*)
          
END_FUNCTION

FUNCTION RES_NTC : REAL
  VAR_INPUT
    T : REAL;
    RN : REAL;
    B : REAL;
  END_VAR

            RES_NTC := RN * EXP(B * (1.0 / (T+273.15) - 0.00335401643468053));



(* revision history

hm 30. dec. 2008	rev 1.0
	original version

hm	11. mar. 2009	rev 1.1
	changed real constants to use dot syntax

*)
          
END_FUNCTION

FUNCTION RES_PT : REAL
  VAR_INPUT
    T : REAL;
    R0 : REAL;
  END_VAR
  VAR CONSTANT
    A : REAL := 0.00390802;
    B : REAL := -5.802E-07;
    C : REAL := -4.2735E-12;
  END_VAR
  VAR
    T2 : REAL;
  END_VAR

            T2 := T * T;

IF T >= 0.0 THEN
	RES_PT := R0 * ( 1.0 + A * T + B * T2);
ELSE
	RES_PT := R0 * ( 1.0 + A * T + B * T2 + C * (T - 100.0) * T2 * T);
END_IF;



(* revision history
hm	4. aug. 2006	rev 1.1
	original version

hm	2. dec 2007	rev 1.2
	changed code for better performance

hm	11. mar. 2009	rev 1.3
	changed real constants to use dot syntax

*)


(*
 Auszug aus DIN 43760 für Pt100

°C		R		°C		R		°C	R			°C		R			°C		R			°C		R

-200 	18,49 	-100 	60,25 	0 	100,00 	100 	138,50 	200 	175,84 	300 	212,02
-195 	20,65 	-95 	62,28 	5 	101,95 	105 	140,39 	205 	177,68 	305 	213,80
-190 	22,80 	-90 	64,30 	10 	103,90 	110 	142,29 	210 	179,51 	310 	215,57
-185 	24,94 	-85 	66,31 	15 	105,85 	115 	144,17 	215 	181,34 	315 	217,35
-180 	27,08 	-80 	68,33 	20 	107,79 	120 	146,06 	220 	183,17 	320 	219,12
-175 	29,20 	-75 	70,33 	25 	109,73 	125 	147,94 	225 	184,99 	325 	220,88
-170 	31,32 	-70 	72,33 	30 	111,67 	130 	149,82 	230 	186,82 	330 	222,65
-165 	33,43 	-65 	74,33 	35 	113,61 	135 	151,70 	235 	188,63 	335 	224,41
-160 	35,33 	-60 	76,33 	40 	115,54 	140 	153,58 	240 	190,45 	340 	226,17
-155 	37,63 	-55 	78,32 	45 	117,47 	145 	155,45 	245 	192,26 	345 	227,92
-150 	39,71 	-50 	80,31 	50 	119,40 	150 	157,31 	250 	194,07 	350 	229,67
-145 	41,79 	-45 	82,29 	55 	121,32 	155 	159,18 	255 	195,88 	355 	231,42
-140 	43,87 	-40 	84,27 	60 	123,24 	160 	161,04 	260 	197,69 	360 	233,17
-135 	45,94 	-35 	86,25 	65 	125,16 	165 	162,90 	265 	199,49 	365 	234,91
-130 	48,00 	-30 	88,22 	70 	127,07 	170 	164,76 	270 	201,29 	370 	236,65
-125 	50,06 	-25 	90,19 	75 	128,98 	175 	166,61 	275 	203,08 	375 	238,39
-120 	52,11 	-20 	92,16 	80 	130,89 	180 	168,46 	280 	204,88 	380 	240,13
-115 	54,15 	-15 	94,12 	85 	132,80 	185 	170,31 	285 	206,67 	385 	241,86
-110 	56,19 	-10 	96,09 	90 	134,70 	190 	172,16 	290 	208,45 	390 	243,59
-105 	58,22 	-5 		98,04 	95 	136,60 	195 	174,00 	295 	210,24 	395 	245,31

*)
(*
revision history


*)
          
END_FUNCTION

FUNCTION RES_SI : REAL
  VAR_INPUT
    T : REAL;
    RS : REAL;
    TS : REAL;
  END_VAR
  VAR CONSTANT
    A : REAL := 0.00764;
    B : REAL := 1.66E-05;
  END_VAR
  VAR
    TX : REAL;
  END_VAR

            TX := T - TS;
RES_SI := RS * ( 1.0 + A * TX + B * TX * TX);

(* revision history
hm	4. aug 2006	rev 1.0
	original version

hm	2. dec 2007	rev 1.1
	changed code for better performance

hm	11. mar. 2009	rev 1.2
	changed real constants to use dot syntax

*)
          
END_FUNCTION

FUNCTION SENSOR_INT : REAL
  VAR_INPUT
    Voltage : REAL;
    Current : REAL;
    RP : REAL;
    RS : REAL;
  END_VAR
  VAR
    RG : REAL;
  END_VAR

            IF current <> 0.0 THEN
	RG := voltage / current;
	SENSOR_INT := RP * ( RG - RS) / ( RP + RS - RG);
END_IF;

(* revisaion history

hm 20.1.2007		rev 1.1
	deleted input R0 which was not needed.

hm	2. dec 2007	rev 1.2
	corrected an error in formula and improoved speed

hm	11. mar. 2009	rev 1.3
	changed real constants to use dot syntax

*)
          
END_FUNCTION

FUNCTION TEMP_NI : REAL
  VAR_INPUT
    Res : REAL;
    R0 : REAL;
  END_VAR

            TEMP_NI := (SQRT(0.30085225 - 2.66E-3 * (R0 - Res)) - 0.5485) * 751.8796992;


(* revision history

hm 24.1.2007		rev 1.1
	deleted unused variable A, B, C

hm 10.9.2007		rev 1.2
	changed accuracy to 0.02 degrees to improove performace

hm 17. 12 2007	rev 1.3
	improovements for better performance and higher accuracy

hm	6. jan 2008	rev 1.4
	further performance improvement

hm	10. mar. 2009	rev 1.5
	removed nested comments

*)


          
END_FUNCTION

FUNCTION TEMP_NTC : REAL
  VAR_INPUT
    RES : REAL;
    RN : REAL;
    B : REAL;
  END_VAR

            IF res > 0.0 THEN
	TEMP_NTC := B * 298.15 / (B + LN(RES / RN) * 298.15) -273.15;
END_IF;


(* revision history

hm 30. dec. 2008	rev 1.0
	original version

hm	11. mar. 2009	rev 1.1
	changed real constants to use dot syntax

*)
          
END_FUNCTION

FUNCTION TEMP_PT : REAL
  VAR_INPUT
    Res : REAL;
    R0 : REAL;
  END_VAR
  VAR CONSTANT
    A : REAL := 0.0039083;
    B : REAL := -5.775E-07;
    accuracy : REAL := 0.01;
  END_VAR
  VAR
    step : REAL := 50;
    X : REAL;
    Y : REAL;
    t1 : REAL;
    pt : POINTER TO DWORD;
  END_VAR

            X := A * R0;
Y := B * R0;
IF Res >= R0 THEN
	t1 := X * X - 4.0 * Y * (R0 - Res);
	IF t1 < 0.0 THEN
		TEMP_PT := 10000.0;
	ELSE
		TEMP_PT := (-X + SQRT(t1)) / (2.0 * Y);
	END_IF;
ELSE
	pt := ADR(step);
	(* since the formula cannot be solved this is a successive approximation *)
	TEMP_PT := -100.0;
	WHILE step > accuracy DO
		(* test if result greater or less *)
		IF RES_PT(TEMP_PT, R0) < res THEN TEMP_PT := TEMP_PT + step; ELSE TEMP_PT := TEMP_PT - step; END_IF;
		pt^ := pt^ - 8388608;  (* this is a super fast divide by 2 method for non floating point CPUs *)
		(* the alternative code: step := step * 0.5; *)
	END_WHILE;
END_IF;

(* revision history

rev 1.1 hm 24.1.2007	
	deleted unused variable C

rev 1.2 hm 10.9.2007
	reduced accuracy to 0.02 to shorten execution time

rev 1.3	hm	2. dec 2007
	changed code for better performance

rev	1.4	hm	23. dec 2007
	avoid a negative square root if input values are wrong

rev 1.5 hm	5. jan 2008
	replaced / 2 with * 0.5 for better performance

hm	31. oct. 2008	rev 1.6
	improved performance

hm	11. mar. 2009	rev 1.7
	changed real constants to use dot syntax

*)

          
END_FUNCTION

FUNCTION TEMP_SI : REAL
  VAR_INPUT
    Res : REAL;
    RS : REAL;
    TS : REAL;
  END_VAR

            TEMP_SI := (-7.64E-3 + SQRT(Res / RS * 6.64E-5 - 0.803E-5)) * 30120.48193 + TS;



(* revision history

hm 24.1.2007		rev 1.1
	the function would only work for TS = 25, now it works for other values of ts.

hm 10.9.2007		rev 1.2
	changed the function to use successive approcimation to avoid an error generated by a sqrt from a negative result.
	changed accuracy to 0.02 degrees to shorten execution time

hm 17. 12 2007	rev 1.3
	improovements for better performance

hm	6. jan 2008	rev 1.4
	further performance improvement

hm	10. mar. 2009	rev 1.5
	removed nested comments

*)
          
END_FUNCTION

FUNCTION_BLOCK _RMP_B
  VAR_INPUT
    DIR : BOOL;  (* true = up *)
    E : BOOL := TRUE;
    TR : TIME;
  END_VAR
  VAR_IN_OUT
    RMP : BYTE;
  END_VAR
  VAR
    tx : TIME;
    tl : TIME;
    tn : TIME;
    init : BOOL;
    last_dir : BOOL;
    start : BYTE;
  END_VAR

            (* read system timer *)
tx := DWORD_TO_TIME(T_PLC_MS());

IF E AND init AND (dir = last_dir) AND (RMP <> SEL(DIR, 0, 255)) AND TR = tn THEN
	RMP := FRMP_B(start, DIR, tx - tl, TR);
ELSE
	init := TRUE;
	tl := tx;
	tn := tr;
	start := RMP;
END_IF;
last_dir := dir;



(* revison history
hm	22. oct. 2008	rev 1.0
	original version

hm	20. nov. 2008	rev 1.1
	set default for E to be TRUE
	added init

hm	19. nov. 2011	rev 1.2
	new code
*)
          
END_FUNCTION_BLOCK

FUNCTION_BLOCK _RMP_NEXT
  VAR_INPUT
    E : BOOL := TRUE;
    IN : BYTE;
    TR : TIME;
    TF : TIME;
    TL : TIME;
  END_VAR
  VAR_OUTPUT
    DIR : BOOL;  (* upwards = TRUE *)
    UP : BOOL;
    DN : BOOL;
  END_VAR
  VAR_IN_OUT
    OUT : BYTE;
  END_VAR
  VAR
    rmx : _RMP_B;
    dirx : TREND_DW;
    t_lock : TP;
    xen : BOOL;
    xdir : BOOL;
  END_VAR

            dirx(X := in);

t_lock(in := FALSE, pt := TL);

IF dirx.TU AND (OUT < IN) THEN
	IF NOT xdir AND xen THEN t_lock(in := TRUE); END_IF;
	xen := TRUE;
	xdir := TRUE;
ELSIF dirx.TD AND (OUT > IN) THEN
	IF xdir AND xen THEN t_lock(in := TRUE); END_IF;
	xen := TRUE;
	xdir := FALSE;
ELSIF xen THEN
	IF (xdir AND (out >= in)) OR (NOT xdir AND (out <= in)) THEN
		xen := FALSE;
		IF tl > t#0s THEN t_lock(IN := TRUE); END_IF;
	END_IF;
END_IF;

IF NOT t_lock.Q AND xen THEN
		UP := XDIR;
		DIR := XDIR;
		DN := NOT XDIR;
ELSE
	UP := FALSE;
	DN := FALSE;
END_IF;

rmx(rmp := OUT, E := E AND (UP OR DN) , dir := DIR, tr := SEL(dir, TF, TR));


(* revison history
hm	23. nov. 2008	rev 1.0
	original version

hm	24. jan. 2009	rev 1.1
	deleted unused vars tmp1, tmp2

hm	20. feb. 2009	rev 1.2
	improved algorithm
	added TL

hm	9. mar. 2009	rev 1.3
	input E was ignored
	removed double assignments

hm	18. jul. 2009	rev 1.4
	improved performance

*)
          
END_FUNCTION_BLOCK

FUNCTION_BLOCK _RMP_W
  VAR_INPUT
    DIR : BOOL;
    E : BOOL := TRUE;
    TR : TIME;
  END_VAR
  VAR_IN_OUT
    RMP : WORD;
  END_VAR
  VAR
    tx : DWORD;
    tl : DWORD;
    step : DINT;
    init : BOOL;
    last_dir : BOOL;
  END_VAR

            tx := T_PLC_MS();
IF E AND init THEN
	(* we need to set tl = tx when direction changes *)
	IF dir XOR last_dir THEN
	 tl := tx;
	 last_dir := dir;
	END_IF;
	(* check_elapsed time and calculate only if necessary *)
	IF tr > t#0s THEN
		step := DWORD_TO_DINT(SHL(tx-tl, 16) / TIME_TO_DWORD(TR));
	ELSE
		step := 65535;
	END_IF;
	IF step > 0 THEN
		(* perform the step on the ramp *)
		tl := tx;
		(* calculate the step response *)
		IF NOT dir THEN step := - step; END_IF;
		rmp := DINT_TO_WORD(LIMIT(0, WORD_TO_DINT(rmp) + step, 65535));
	END_IF;
ELSE
	tl := tx;
	init := TRUE;
END_IF;


(* revison history
hm	22. oct. 2008	rev 1.0
	original version

hm	20. nov. 2008	rev 1.1
	set default for E to be TRUE
	added init

*)
          
END_FUNCTION_BLOCK

FUNCTION_BLOCK GEN_PULSE
  VAR_INPUT
    ENQ : BOOL := TRUE;
    PTH : TIME;
    PTL : TIME;
  END_VAR
  VAR_OUTPUT
    Q : BOOL;
  END_VAR
  VAR
    tx : TIME;
    tn : TIME;
    init : BOOL;
  END_VAR

            
IF enq THEN
	tx := DWORD_TO_TIME(T_PLC_MS());
	IF NOT init THEN init := TRUE; tn := tx; END_IF;
	IF tx - tn >= SEL(Q, PTL, PTH) THEN
		Q := NOT Q;
		tn := tn + SEL(Q, PTL, PTH);
	END_IF;
ELSE
	Q := FALSE;
	init := FALSE;
END_IF;


(* revision history
hm	29. jun. 2008	rev 1.0
	original version

hm	23. nov. 2008	rev 1.1
	set default for enq to be true

hm	18. jul. 2009	rev 1.2
	improved performance

hm	13. nov. 2009	rev 1.3
	corrected error

hm	16. feb. 2011	rev 1.4
	corrected an error when timer overflows

*)
          
END_FUNCTION_BLOCK

FUNCTION_BLOCK GEN_PW2
  VAR_INPUT
    ENQ : BOOL;
    TH1 : TIME;
    TL1 : TIME;
    TH2 : TIME;
    TL2 : TIME;
    TS : BOOL;
  END_VAR
  VAR_OUTPUT
    Q : BOOL;
    TH : TIME;
    TL : TIME;
  END_VAR
  VAR
    t_high : TIME;
    t_low : TIME;
    tx : TIME;
    start : TIME;
    init : BOOL;
    et : TIME;
  END_VAR

            (* read system timer *)
tx := DWORD_TO_TIME(T_PLC_MS());

(* startup initialization *)
IF NOT init THEN
	start := tx;
	init := TRUE;
	TH := T#0s;
	TL := T#0s;
END_IF;

(* timing selection *)
IF TS THEN
	t_high := TH2;
	t_low := TL2;
ELSE
	t_high := TH1;
	t_low := TL1;
END_IF;

(* normal operation *)
IF ENQ THEN
	et := tx - start;
	IF NOT Q THEN
		IF et >= t_low THEN
			Q := TRUE;
			start := tx;
			TL := T#0s;
		ELSE
			TL := et;
		END_IF;
	ELSE
		IF et >= t_high THEN
			Q := FALSE;
			start := tx;
			TH := T#0s;
		ELSE
			TH := et;
		END_IF;
	END_IF;
ELSE
	Q := FALSE;
	TH := T#0s;
	TL := T#0s;
	start := tx;
END_IF;



(* revision history
hm	26. sep. 2008	rev 1.0
	original version

hm	14. mar. 2009	rev 1.1
	removed double assignments

*)
          
END_FUNCTION_BLOCK

FUNCTION_BLOCK GEN_RDM
  VAR_INPUT
    PT : TIME;
    AM : REAL := 1;
    OS : REAL;
  END_VAR
  VAR_OUTPUT
    Q : BOOL;
    Out : REAL;
  END_VAR
  VAR
    tx : TIME;
    last : TIME;
    init : BOOL;
  END_VAR

            (* read system time and prepare input data *)
tx := DWORD_TO_TIME(T_PLC_MS()) - last;

(* init section *)
IF NOT init THEN
	init := TRUE;
	last := tx;
	tx := t#0s;
END_IF;

(* add last if one cycle is finished *)
IF tx >= pt THEN
	last := last + pt;
	tx := tx - pt;

	(* generate output signal *)
	out := am * (RDM(0) - 0.5) + os;
	q := TRUE;
ELSE
	q := FALSE;
END_IF;

(* revision history

hm	7.2.2007		rev 1.0
	original version

hm	16.9.2007		rev 1.1
	changes time() to T_plc_ms() for compatibility reasons

*)

          
END_FUNCTION_BLOCK

FUNCTION_BLOCK GEN_RDT
  VAR_INPUT
    Enable : BOOL := TRUE;
    Min_Time_ms : TIME := TIME#1s0ms;  (* min Taktzeit *)
    Max_Time_ms : TIME := TIME#1s200ms;  (* Max Taktzeit *)
    TP_Q : TIME := TIME#100ms;  (* Zeit Ausgang auf TRUE *)
  END_VAR
  VAR_OUTPUT
    xQ : BOOL;
  END_VAR
  VAR
    tonRDMTimer : TON;  (* Zeitbaustein Taktgenerator *)
    tof_xQ : TOF;  (* Ausschaltverzögerung Taktgenerator *)
    tRDMTime : TIME;  (* Sollzeit *)
    rRDMTime : REAL;  (* Zufalswert Timer *)
  END_VAR

            tonRDMTimer ( IN:= Enable , PT:= tRDMTime );
tof_xQ ( IN:= tonRDMTimer.Q , PT:= TP_Q );
XQ := tof_xq.Q;
IF tonRDMTimer.Q THEN
		 xQ := TRUE ;
		 rRDMTime := RDM ( last:= rRDMTime ) ;
		 tRDMTime := REAL_TO_TIME ( rRDMTime * DINT_TO_REAL(TIME_TO_DINT( Max_Time_ms - Min_Time_ms ) + TIME_TO_DINT(Min_Time_ms ))) ;
		 tonRDMTimer ( IN:= FALSE );
END_IF;

(* revision history
J. Schohaus	19. nov 2007	rev 1.0
	origial version

hm	16. mar. 2008			rev 1.1
	added type conversion to avoid warnings under codesys 3.0
*)
          
END_FUNCTION_BLOCK

FUNCTION_BLOCK GEN_RMP
  VAR_INPUT
    PT : TIME := TIME#1s0ms;
    AM : REAL := 1;
    OS : REAL;
    DL : REAL;
  END_VAR
  VAR_OUTPUT
    Q : BOOL;
    OUT : REAL;
  END_VAR
  VAR
    tx : TIME;
    last : TIME;
    init : BOOL;
    temp : REAL;
    ltemp : REAL;
  END_VAR

            (* read system time and prepare input data *)
tx := DWORD_TO_TIME(T_PLC_MS()) - last;
DL := MODR(dl,1.0);
IF dl < 0.0 THEN dl := 1.0 - dl; END_IF;

(* init section *)
IF NOT init THEN
	init := TRUE;
	last := tx;
	tx := t#0s;
END_IF;

(* add last if one cycle is finished *)
IF tx >= pt THEN
	last := last + pt;
	tx := tx - pt;
END_IF;

(* generate sine wave *)
ltemp := temp;
IF pt > t#0s THEN temp := FRACT(TIME_TO_REAL(tx + MULTIME(pt, dl)) / TIME_TO_REAL(pt)); END_IF;
out := am * temp + os;

(* boolean output Q *)
Q := temp < ltemp;

(* revision history
hm	3. mar 2007		rev 1.0
	original version

hm	17 sep 2007		rev 1.1
	replaced time() with t_plc_ms for compatibilitx reasons

hm	27. nov 2007	rev 1.2
	avoid divide by 0 when pt = 0

ks	26. oct. 2008	rev 1.3
	code optimization

hm	10. mar. 2009	rev 1.4
	changed real constants to use dot syntax
*)
          
END_FUNCTION_BLOCK

FUNCTION_BLOCK GEN_SIN
  VAR_INPUT
    PT : TIME;
    AM : REAL := 1;
    OS : REAL;
    DL : REAL;
  END_VAR
  VAR_OUTPUT
    Q : BOOL;
    Out : REAL;
  END_VAR
  VAR
    tx : TIME;
    last : TIME;
    init : BOOL;
    temp : REAL;
  END_VAR

            (* read system time and prepare input data *)
tx := DWORD_TO_TIME(T_PLC_MS()) - last;
DL := MODR(dl,1.0);
IF dl < 0.0 THEN dl := 1.0 - dl; END_IF;

(* init section *)
IF NOT init THEN
	init := TRUE;
	last := tx;
	tx := t#0s;
END_IF;

(* add last if one cycle is finished *)
IF tx >= pt THEN
	last := last + pt;
	tx := tx - pt;
END_IF;

(* generate sine wave *)
IF pt > t#0s THEN temp := SIN(math.PI2 * DWORD_TO_REAL(TIME_TO_DWORD(tx + MULTIME(pt, dl))) / DWORD_TO_REAL(TIME_TO_DWORD(pt))); END_IF;
out := am * 0.5 *  temp + os;

(* boolean output Q *)
q := NOT SIGN_R(temp);

(* revision history
hm	22. jan 2007	rev 1.0
	original version

hm	17 sep 2007	rev 1.1
	replaced time() with t_plc_ms for compatibilitx reasons

hm	27. nov 2007	rev 1.2
	avoid divide by 0 when pt = 0

hm	6. jan 2008		rev 1.3
	improved performance

hm	16. mar. 2008	rev 1.4
	added type conversion to avoid warnings under codesys 3.0

hm	18. oct. 2008	rev 1.5
	using math constants

hm	11. mar. 2009	rev 1.6
	changed real constants to use dot syntax

*)
          
END_FUNCTION_BLOCK

FUNCTION_BLOCK GEN_SQR
  VAR_INPUT
    PT : TIME;
    AM : REAL := 1;
    OS : REAL;
    DC : REAL := 0.5;
    DL : REAL;
  END_VAR
  VAR_OUTPUT
    Q : BOOL;
    Out : REAL;
  END_VAR
  VAR
    tx : TIME;
    last : TIME;
    init : BOOL;
  END_VAR

            (* check dc = 1 or 0 *)
IF dc = 0.0 THEN
	out := -am * 0.5 + os;
	Q := FALSE;
	RETURN;
ELSIF dc = 1.0 THEN
	out := am * 0.5 + os;
	Q := TRUE;
	RETURN;
END_IF;

(* read system time and prepare input data *)
tx := DWORD_TO_TIME(T_PLC_MS()) - last;
DL := MODR(dl,1.0);
IF dl < 0.0 THEN dl := 1.0 - dl; END_IF;
dc := MODR(dc,1.0);
IF dc < 0.0 THEN dc := 1.0 - dc; END_IF;

(* init section *)
IF NOT init THEN
	init := TRUE;
	last := tx;
	tx := t#0s;
END_IF;

(* add last if one cycle is finished *)
IF tx >= pt THEN
	last := last + pt;
	tx := tx - pt;
END_IF;

(* check if falling or rising edge first *)
IF MULTIME(pt, dl + dc) >= pt THEN
	(* generate falling edge *)
	IF tx >= MULTIME(pt, dl + dc - 1) THEN
		out := -am * 0.5 + os;
		Q := FALSE;
	END_IF;
	(* generate rising edge *)
	IF tx >= MULTIME(pt, dl) THEN
		out := am * 0.5 + os;
		Q := TRUE;
	END_IF;
ELSE
	(* generate rising edge first *)
	IF tx >= MULTIME(pt, dl) THEN
		out := am * 0.5 + os;
		Q := TRUE;
	END_IF;
	(* generate falling edge *)
	IF tx >= MULTIME(pt, dl + dc) THEN
		out := -am * 0.5 +os;
		Q := FALSE;
	END_IF;
END_IF;

(* revision history

hm	12. feb 2007	rev 1.1
	added default value for dc = 0.5

hm	17 sep 2007	rev 1.2
	replaced time() with t_plc_ms for compatibilitx reasons

hm	6. jan 2008	rev 1.3
	improved performance

hm	11. mar. 2009	rev 1.4
	changed real constants to use dot syntax
	set default amplitude to 1.0

*)

          
END_FUNCTION_BLOCK

FUNCTION_BLOCK PWM_DC
  VAR_INPUT
    F : REAL;
    DC : REAL;
  END_VAR
  VAR_OUTPUT
    Q : BOOL;
  END_VAR
  VAR
    clk : CLK_PRG;
    pulse : TP_X;
    tmp : REAL;
  END_VAR

            IF F > 0.0 THEN
	tmp := 1000.0 / F;
	CLK(PT := REAL_TO_TIME(tmp));
	Pulse(in := clk.Q, pt := REAL_TO_TIME(tmp * DC));
	Q := pulse.Q;
END_IF;

(* revision history

hm	25. feb 2007	rev 1.1
	recoded in st for better performance and better portability

hm	27. nov 2007	rev 1.2
	avoid divide by 0 when F = 0

hm	19. oct. 2008	rev 1.3
	changed type TP_R to TP_X because of name change
	improved performance

hm	11. mar. 2009	rev 1.4
	changed real constants to use dot syntax

*)
          
END_FUNCTION_BLOCK

FUNCTION_BLOCK PWM_PW
  VAR_INPUT
    F : REAL;
    PW : TIME;
  END_VAR
  VAR_OUTPUT
    Q : BOOL;
  END_VAR
  VAR
    clk : CLK_PRG;
    pulse : TP_X;
  END_VAR

            IF F > 0.0 THEN
	CLK(PT := REAL_TO_TIME(1000.0 / F));
	Pulse(in := clk.Q, pt := pw);
	Q := pulse.Q;
END_IF;

(* revision history

hm	25. feb 2007	rev 1.1
	recoded in st for better performance and better portability

hm	27. nov 2007	rev 1.2
	avoid divide by 0 when F = 0

hm	9. dec 2007		rev 1.3
	corrected an error with F = 0

hm	19. oct. 2008	rev 1.4
	changed type tp_r to TP_x brecause of name change

hm	11. mar. 2009	rev 1.5
	changed real constants to use dot syntax

*)
          
END_FUNCTION_BLOCK

FUNCTION_BLOCK RMP_B
  VAR_INPUT
    SET : BOOL;
    PT : TIME;
    E : BOOL := TRUE;
    UP : BOOL := TRUE;
    RST : BOOL;
  END_VAR
  VAR_OUTPUT
    OUT : BYTE;
    BUSY : BOOL;
    HIGH : BOOL;
    LOW : BOOL;
  END_VAR
  VAR
    rmp : _RMP_B;
  END_VAR

            (* generate ramp *)
rmp(dir := UP, E := E, TR := PT, rmp := out);

(* set or reset operation *)
IF RST THEN
	out := 0;
ELSIF SET THEN
	out := 255;
END_IF;

(* checks for outputs stable and reset or set busy flag *)
low := out = 0;
high := out = 255;
busy := NOT (low OR high) AND E;


(* revision history

hm 5.10.2006	rev 1.1
	added busy output
hm 17.1.2007	rev 1.2
	renamed input ud to up for better usability
	deleted unused variable step

hm	17.9.2007		rev 1.3
	replaced time() with t_plc_ms() for compatibility reasons

hm	28. sep 2007	rev 1.4
	added outputs on and off
	busy is now disabled while en is false
	new coding for higher accuracy and performance

hm	5. oct 2007	rev 1.5
	added statements to allow for PT to be t#0s output jumps to max or min immediately

hm	25. dec 2007	rev 1.6
	improved code for better performance

hm	16. oct. 2008	rev 1.7
	improved code for better performance

hm	18. oct. 2008	rev 1.8
	added type conversion to avoid warnings
	changed input en to e for compatibility reasons

hm	23. oct. 2008	REV 	2.0
	new code using _RMP_B

*)
          
END_FUNCTION_BLOCK

FUNCTION_BLOCK RMP_SOFT
  VAR_INPUT
    IN : BOOL;
    VAL : BYTE;
    {attribute 'input_constant'}
    PT_ON : TIME;
    {attribute 'input_constant'}
    PT_OFF : TIME;
  END_VAR
  VAR_OUTPUT
    OUT : BYTE;
  END_VAR
  VAR
    rmp : _RMP_B;
    tmp : BYTE;
  END_VAR

            tmp := SEL(in, 0, val);
IF tmp > out THEN
	(* we need to ramp down *)
	rmp(dir := TRUE, E := TRUE, TR := PT_ON, rmp := out);
	(* make sure out does not surpass tmp *)
	out := MIN(out, tmp);
ELSIF tmp < out THEN
	(* we need to ramp up *)
	rmp(dir := FALSE, E := TRUE, TR := PT_OFF, rmp := out);
	(* make sure out does not surpass tmp *)
	out := MAX(out, tmp);
ELSE
	(* no ramp necessary *)
	rmp(E := FALSE, rmp := out);
END_IF;


(* revision history

hm 22.1.2007	rev 1.1
	deleted unused variables X1 and I, X2 and X3

hm	17.9.2007	rev 1.2
	replaced time() with t_plc_ms() for compatibility reasons

hm	26. oct. 2008	2.0
	new code using _rmp_b
*)

          
END_FUNCTION_BLOCK

FUNCTION_BLOCK RMP_W
  VAR_INPUT
    SET : BOOL;
    PT : TIME;
    E : BOOL := TRUE;
    UP : BOOL := TRUE;
    RST : BOOL;
  END_VAR
  VAR_OUTPUT
    out : WORD;
    busy : BOOL;
    high : BOOL;
    low : BOOL;
  END_VAR
  VAR
    rmp : _RMP_W;
  END_VAR

            (* generate ramp *)
rmp(dir := UP, E := E, TR := PT, rmp := out);

(* set or reset operation *)
IF RST THEN
	out := 0;
ELSIF SET THEN
	out := 65535;
END_IF;

(* checks for outputs stable and reset or set busy flag *)
low := out = 0;
high := out = 65535;
busy := NOT (low OR high) AND E;


(* revision history:

hm 4.10.2006		rev 1.1
	added the busy output which signals that the ramp is running.

hm 22.1.2007		rev 1.2
	deleted unused variable step

hm	17.9.2007		rev 1.3
	replaced time() with t_plc_ms() for compatibility reasons

hm	28. sep 2007	rev 1.4
	added outputs on and off
	busy is now disabled while en is false
	new coding for higher accuracy and performance

hm	5. oct 2007	rev 1.5
	added statements to allow for PT to be t#0s output jumps to max or min immediately

hm	2. dec 2007	rev 1.6
	corrected an error in calculation of step response

hm	25. dec 2007	rev 1.7
	corrected an error while step response was too slow for fast rise times

hm	16. oct. 2008	rev 1.8
	improved performance

hm	18. oct. 2008	rev 1.9
	renamed inout EN to E for compatibility reasons

hm	23. oct. 2008	rev 2.0
	new code using _RMP_W
*)

          
END_FUNCTION_BLOCK

FUNCTION AIN : REAL
  VAR_INPUT
    in : DWORD;
    {attribute 'input_constant'}
    Bits : BYTE;
    {attribute 'input_constant'}
    sign : BYTE := 255;
    {attribute 'input_constant'}
    low : REAL;
    {attribute 'input_constant'}
    high : REAL := 10;
  END_VAR
  VAR CONSTANT
    ff : DWORD := 16#FFFFFFFF;
  END_VAR
  VAR
    temp1 : DWORD;
    temp2 : DWORD;
    sx : BOOL;
  END_VAR

            (* extract the sign bit *)
IF sign < 32 THEN
	temp1 := SHR(in,sign);
	sx := temp1.0;
ELSE
	sx := FALSE;
END_IF;
temp1 := SHR(ff, 32-bits);
temp2 := in AND temp1;
AIN := (high - low) * DWORD_TO_REAL(temp2) / DWORD_TO_REAL(temp1) + low;
IF sx THEN AIN := -AIN; END_IF;

(* revision history
hm 18.8.2006	rev 1.1
	fixed an error with low value negative and high value 0.

hm 19.1.2007	rev 1.2
	fixed an error with sign bit.

hm	13.9.2007	rev 1.3
	changed code to avoid warning under codesys 2.8.1

hm	2. dec 2007	rev 1.4
	changed code for better performance

hm	16. mar 2008	rev 1.5
	added type conversions to avoid warnings under codesys 30
*)
          
END_FUNCTION

FUNCTION_BLOCK AIN1
  VAR_INPUT
    in : DWORD;
    {attribute 'input_constant'}
    sign_bit : INT := 255;
    {attribute 'input_constant'}
    error_bit : INT := 255;
    {attribute 'input_constant'}
    error_code_en : BOOL;
    {attribute 'input_constant'}
    error_code : DWORD;
    {attribute 'input_constant'}
    overflow_bit : INT := 255;
    {attribute 'input_constant'}
    overflow_code_en : BOOL;
    {attribute 'input_constant'}
    overflow_code : DWORD;
    {attribute 'input_constant'}
    Bit_0 : INT;
    {attribute 'input_constant'}
    Bit_N : INT := 31;
    {attribute 'input_constant'}
    out_min : REAL;
    {attribute 'input_constant'}
    out_max : REAL := 10;
    {attribute 'input_constant'}
    code_min : DWORD;
    {attribute 'input_constant'}
    code_max : DWORD := 16#FFFFFFFF;
    {attribute 'input_constant'}
    error_output : REAL;
    {attribute 'input_constant'}
    overflow_output : REAL := 10;
  END_VAR
  VAR_OUTPUT
    out : REAL;
    sign : BOOL;
    error : BOOL;
    overflow : BOOL;
  END_VAR
  VAR
    tB : DWORD;
  END_VAR

            (* extract error bit *)
error := ((SHR(in,error_bit) AND 16#0000_0001) = 1) OR (error_code_en AND error_code = in);
IF error THEN
	out := error_output;
	RETURN;
END_IF;

(* strip off the data input *)
tb := SHR(SHL(in, 31 - bit_N), 31 - bit_N + Bit_0);

(* extract overflow bit *)
overflow := ((SHR(in,overflow_bit) AND 16#0000_0001) = 1) OR (overflow_code_en AND overflow_code = in) OR (tb < code_min OR tb > code_max);
IF overflow THEN
	out := overflow_output;
	RETURN;
END_IF;

(* extract sign bit *)
sign := (SHR(in,sign_bit) AND 16#0000_0001) = 1;

(* convert in to out *)
out := (DWORD_TO_REAL(tb - code_min) * (out_max - out_min) / DWORD_TO_REAL(code_max - code_min) + out_min);
IF sign THEN out := out * -1.0; END_IF;



(* revision history
hm	23. feb 2008	rev 1.0
	original version

hm	16. mar 2008	rev 1.1
	added type conversions to avoid warnngs under codesys 30

hm	22. apr. 2008	rev 1.2
	corrected error in formula when code_min was set
	corrected error when sign bit was used
	optimized code for better performance

hm	10. mar. 2009	rev 1.3
	real constants updated to new systax using dot

*)
          
END_FUNCTION_BLOCK

FUNCTION AOUT : DWORD
  VAR_INPUT
    in : REAL;
    {attribute 'input_constant'}
    Bits : BYTE;
    {attribute 'input_constant'}
    sign : BYTE := 255;
    {attribute 'input_constant'}
    low : REAL;
    {attribute 'input_constant'}
    high : REAL := 10;
  END_VAR
  VAR CONSTANT
    ff : DWORD := 2#1;
  END_VAR
  VAR
    in2 : REAL;
    sx : BOOL;
  END_VAR

            (* if sign bit is defined *)
IF sign < 32 THEN
	sx := sign_R(in);
	in2 := ABS(in);
ELSE
	in2 := in;
END_IF;

(* begrenze in auf die zulässigen werte *)
in2 := LIMIT(low, in2, high);

(* Berechne den Ausgangswert *)
Aout := REAL_TO_DWORD((in2 - low) / (high - low) * DWORD_TO_REAL(SHL(ff,bits) -1));
IF sx THEN Aout := SHL(ff,sign) OR Aout; END_IF;

(*
revision history

hm 18.1.2007		rev 1.1
	renamed Modul to aout.
	changed Output to 32 Bit max.
	corrected error with sign bit.

hm	13.9.2007		rev 1.2
	changed code to avoid warning under codesys 2.8.1

hm	2. dec 2007		rev 1.3
	changed code for better performance

hm	23. feb 2008	rev 1.4
	changed code for better performance
*)
          
END_FUNCTION

FUNCTION AOUT1 : DWORD
  VAR_INPUT
    in : REAL;
    {attribute 'input_constant'}
    Bit_0 : INT;
    {attribute 'input_constant'}
    Bit_N : INT := 31;
    {attribute 'input_constant'}
    sign : INT := 255;
    {attribute 'input_constant'}
    low : REAL;
    {attribute 'input_constant'}
    high : REAL := 10;
  END_VAR
  VAR CONSTANT
    ff : DWORD := 2#1;
  END_VAR
  VAR
    sx : BOOL;
    in2 : REAL;
  END_VAR

            (* if sign bit is defined *)
IF sign < 32 THEN
	sx := SIGN_R(in);
	in2 := ABS(in);
ELSE
	in2 := in;
END_IF;

(* begrenze in auf die zulässigen werte *)
in2 := LIMIT(low, in2, high);

(* Berechne den Ausgangswert *)
AOUT1 := SHL(REAL_TO_DWORD((in2 - low) / (high - low) * DWORD_TO_REAL(SHL(ff,bit_n - Bit_0 + 1) -1)),Bit_0);
IF sx THEN AOUT1 := SHL(ff,sign) OR AOUT1; END_IF;


(* revision history
hm	23. feb 2008	rev 1.0
	original version

*)
          
END_FUNCTION

FUNCTION BYTE_TO_RANGE : REAL
  VAR_INPUT
    X : BYTE;
    low : REAL;
    high : REAL;
  END_VAR

            BYTE_TO_RANGE := (high - low) * X / 255.0 + low;


(* revision history
hm	9. jan 2008		rev 1.0
	original version

*)

          
END_FUNCTION

FUNCTION_BLOCK DELAY
  VAR_INPUT
    IN : REAL;
    N : INT;
    RST : BOOL;
  END_VAR
  VAR_OUTPUT
    OUT : REAL;
  END_VAR
  VAR
    buf : ARRAY[0..31] OF REAL;
    i : INT;
    init : BOOL;
    stop : INT;
  END_VAR

            stop := LIMIT(0,N,32) - 1;
IF rst OR NOT init THEN
	init := TRUE;
	FOR i := 0 TO stop DO buf[i] := in; END_FOR;
	out := in;
	i := 0;
ELSIF stop < 0 THEN
	out := in;
ELSE
	out := buf[i];
	buf[i] := in;
	i := INC1(i, N);
END_IF;



(* revision history
hm 1.10.2006		rev 1.1
	corrected error in buffer management

hm 19.1.2007		rev 1.2
	changed reset to load the value of in instead of 0

hm	27. oct. 2008	rev 1.3
	improved performance

hm	23. feb.2009	rev 1.4
	corrected an index problem

hm	23. mar. 2009	rev 1.5
	corrected non standard write to input N

*)
          
END_FUNCTION_BLOCK

FUNCTION_BLOCK DELAY_4
  VAR_INPUT
    in : REAL;
  END_VAR
  VAR_OUTPUT
    out1 : REAL;
    out2 : REAL;
    out3 : REAL;
    out4 : REAL;
  END_VAR
  VAR
    temp : REAL;
  END_VAR

            out4 := out3;
out3 := out2;
out2 := out1;
out1 := temp;
temp := in;

(* revision history

hm 19.1.2007	rev 1.1
	added variable temp to add 1 delay  for q1

*)
          
END_FUNCTION_BLOCK

FUNCTION_BLOCK FADE
  VAR_INPUT
    IN1 : REAL;
    IN2 : REAL;
    F : BOOL;
    TF : TIME;
    rst : BOOL;
  END_VAR
  VAR_OUTPUT
    Y : REAL;
  END_VAR
  VAR
    rmx : RMP_W;
  END_VAR

            rmx(rst := rst AND NOT F, set := rst AND F, pt := TF, up := F);
Y := (in2 - In1) / 65535.0 * WORD_TO_REAL(rmx.out) + in1;


(* code for rev 1.1
IF rst THEN
	rmx(set := F, rst := NOT F);
ELSIF F AND (NOT rmx.high) THEN
	rmx(PT := TF, UP := TRUE, e := TRUE, rst := FALSE, set := FALSE);
ELSIF (NOT F) AND (NOT rmx.low) THEN
	rmx(PT := TF, UP := FALSE, e := TRUE, rst := FALSE, set := FALSE);
ELSE
	rmx(e := FALSE, rst := FALSE, set := FALSE);
END_IF;
Y := (WORD_TO_REAL(rmx.out) * in1 + WORD_TO_REAL(FF - rmx.out) * IN2) / FF;
*)


(* revision history
hm	26. dec 2007	rev 1.0
	original version

hm	18. oct. 2008	rev 1.1
	improved performance
	changed calls for rmp_w because rmp_w has chaged

hm	17. dec. 2008	rev 1.2
	function of input f was inverted

hm	24. jan. 2009	rev 1.3
	delted unused var FF
*)
          
END_FUNCTION_BLOCK

FUNCTION_BLOCK FILTER_DW
  VAR_INPUT
    X : DWORD;
    T : TIME;
  END_VAR
  VAR_OUTPUT
    Y : DWORD;
  END_VAR
  VAR
    last : DWORD;
    tx : DWORD;
    init : BOOL;
    Yi : REAL;
  END_VAR

            (* read system time *)
tx := T_PLC_MS();

(* startup initialisation *)
IF NOT init OR T = t#0s THEN
	init := TRUE;
	Yi := DWORD_TO_REAL(X);
ELSE
	Yi := Yi + (DWORD_TO_REAL(X) - DWORD_TO_REAL(Y)) * DWORD_TO_REAL(tx - last) / TIME_TO_REAL(T);
END_IF;
last := tx;

Y := REAL_TO_DWORD(Yi);



(*
hm 10. oct. 2008	rev 1.0
	original version

hm	3. nov. 2008	REV 1.1
	corrected an overflow problem
*)
          
END_FUNCTION_BLOCK

FUNCTION_BLOCK FILTER_I
  VAR_INPUT
    X : INT;
    T : TIME;
  END_VAR
  VAR_OUTPUT
    Y : INT;
  END_VAR
  VAR
    Yi : DINT;
    last : DWORD;
    tx : DWORD;
    init : BOOL;
  END_VAR

            (* read system time *)
tx := T_PLC_MS();

(* startup initialisation *)
IF NOT init OR T = t#0s THEN
	init := TRUE;
	Yi := INT_TO_DINT(X) * 1000;
ELSE
	(* to increase accuracy of the filter we calculate internal Yi wich is Y * 1000 *)
	Yi := Yi + INT_TO_DINT(X - Y) * DWORD_TO_DINT(tx - last) * 1000 / TIME_TO_DINT(T);
END_IF;
last := tx;
Y := DINT_TO_INT(yi / 1000);



(*
hm 8. nov. 2008	rev 1.0
	original version

*)
          
END_FUNCTION_BLOCK

FUNCTION_BLOCK FILTER_MAV_DW
  VAR_INPUT
    X : DWORD;
    N : UINT;
    RST : BOOL;
  END_VAR
  VAR_OUTPUT
    Y : DWORD;
  END_VAR
  VAR
    init : BOOL;
    buffer : ARRAY[0..31] OF DWORD;
    i : INT;
    tmp : INT;
  END_VAR

            (* limit N to size of buffer *)
N := MIN(N, 32);

(* startup initialisation *)
IF NOT init OR rst OR N = 0 THEN
	init := TRUE;
	tmp := UINT_TO_INT(N)-1;
	FOR i := 0 TO tmp DO
		buffer[i] := X;
	END_FOR;
	Y := X;
ELSE
	tmp := UINT_TO_INT(N);
	i := INC1(i, tmp);
	Y := Y + (X - buffer[i]) / N;
	buffer[i] := X;
END_IF;




(*
hm 13. oct. 2008	rev 1.0
	original version

hm	27. oct. 2008	rev 1.1
	added typecast to avoid warnings

hm	24. nov. 2008	rev 1.2
	added typecasts to avoid warnings
	avoid divide by 0 if N = 0

hm	23. feb. 2009	rev 1.3
	limit N to max array size

*)
          
END_FUNCTION_BLOCK

FUNCTION_BLOCK FILTER_MAV_W
  VAR_INPUT
    X : WORD;
    N : UINT;
    RST : BOOL;
  END_VAR
  VAR_OUTPUT
    Y : WORD;
  END_VAR
  VAR
    init : BOOL;
    buffer : ARRAY[0..31] OF WORD;
    i : INT;
    tmp : INT;
  END_VAR

            (* limit N to size of buffer *)
N := MIN(N, 32);

(* startup initialisation *)
IF NOT init OR rst OR N = 0 THEN
	init := TRUE;
	tmp := UINT_TO_INT(N) - 1;
	FOR i := 0 TO tmp DO
		buffer[i] := X;
	END_FOR;
	Y := X;
ELSE
	tmp := UINT_TO_INT(N);
	i := INC1(i, tmp);
	Y := Y + (X - buffer[i]) / N;
	buffer[i] := X;
END_IF;



(*
hm 13. oct. 2008	rev 1.0
	original version

hm	18. oct. 2008	rev 1.1
	added typecast to avoid warnings

hm	24. nov. 2008	rev 1.2
	added typecasts to avoid warnings
	avoid devide by 0 if N = 0

hm	23. feb. 2009	rev 1.3
	limit N to max array size

*)
          
END_FUNCTION_BLOCK

FUNCTION_BLOCK FILTER_W
  VAR_INPUT
    X : WORD;
    T : TIME;
  END_VAR
  VAR_OUTPUT
    Y : WORD;
  END_VAR
  VAR
    last : DWORD;
    tx : DWORD;
    init : BOOL;
    tmp : DWORD;
  END_VAR

            (* read system time *)
tx := T_PLC_MS();

(* startup initialisation *)
IF NOT init OR T = T#0s THEN
	init := TRUE;
	last := tx;
	Y := X;
ELSIF Y = X THEN
	last := tx;
ELSE
	tmp :=  WORD_TO_DWORD(X - Y) * (tx - last) / TIME_TO_DWORD(T);
	IF tmp <> 0 THEN
		Y := DINT_TO_WORD(WORD_TO_DINT(Y) + DWORD_TO_DINT(tmp));
		last := tx;
	END_IF;
END_IF;

(*
hm 10. oct. 2008	rev 1.0
	original version

hm	3. nov. 2008	rev 1.1
	fixed overflow problem in formula

hm	25. jan. 2011	rev 1.2
	fixed error in formula
*)
          
END_FUNCTION_BLOCK

FUNCTION_BLOCK FILTER_WAV
  VAR_INPUT
    X : REAL;
    W : ARRAY[0..15] OF REAL;
    RST : BOOL;
  END_VAR
  VAR_OUTPUT
    Y : REAL;
  END_VAR
  VAR
    init : BOOL;
    buffer : ARRAY[0..15] OF REAL;
    i : INT;
    n : INT;
  END_VAR

            (* startup initialisation *)
IF NOT init OR rst THEN
	init := TRUE;
	FOR i := 0 TO 15 DO
		buffer[i] := X;
	END_FOR;
	i := 15;
	Y := X;
ELSE
	i := INC1(i, 16);
	buffer[i] := X;
END_IF;

(* calculate the weighted average *)
Y := 0.0;
FOR n := 0 TO 15 DO
	Y := buffer[i] * W[n] + Y;
	i := DEC1(i, 16);
END_FOR;


(*
hm 	14. oct. 2008	rev 1.0
	original version

hm	27. oct. 2008	rev 1.1
	changed _DEC and _INC to DEC1 and INC1

hm	10. mar. 2009	rev 1.2
	real constants updated to new systax using dot

*)

          
END_FUNCTION_BLOCK

FUNCTION MIX : REAL
  VAR_INPUT
    A : REAL;
    B : REAL;
    M : REAL;
  END_VAR

            MIX := (1.0 - M) * A + M * B;

(* revision history
hm	19. Nov 2007	rev 1.0
	original version

hm	10. mar 2009	rev 1.1
	real constants updated to new systax using dot

*)
          
END_FUNCTION

FUNCTION MUX_R2 : REAL
  VAR_INPUT
    IN0 : REAL;
    IN1 : REAL;
    A : BOOL;
  END_VAR

            MUX_R2 := SEL(A, IN0, IN1);


(* revision history
hm	19. jan. 2007	rev 1.0
	original version

hm	16. oct. 2008	rev 1.1
	improved performance


*)
          
END_FUNCTION

FUNCTION MUX_R4 : REAL
  VAR_INPUT
    IN0 : REAL;
    IN1 : REAL;
    IN2 : REAL;
    IN3 : REAL;
    A0 : BOOL;
    A1 : BOOL;
  END_VAR

            IF A1 THEN
	MUX_R4 := SEL(A0, IN2, IN3);
ELSE
	MUX_R4 := SEL(A0, IN0, IN1);
END_IF;



(* revision history
hm	19. jan 2007	rev 1.0
	original version

hm	16. oct. 2008	rev 1.1
	improved performance
*)
          
END_FUNCTION

FUNCTION OFFSET : REAL
  VAR_INPUT
    X : REAL;
    O1 : BOOL;
    O2 : BOOL;
    O3 : BOOL;
    O4 : BOOL;
    D : BOOL;
    {attribute 'input_constant'}
    Offset_1 : REAL;
    {attribute 'input_constant'}
    Offset_2 : REAL;
    {attribute 'input_constant'}
    Offset_3 : REAL;
    {attribute 'input_constant'}
    Offset_4 : REAL;
    {attribute 'input_constant'}
    default : REAL;
  END_VAR

            IF D THEN OFFSET := default; ELSE OFFSET := X; END_IF;
IF O1 THEN OFFSET := OFFSET + offset_1; END_IF;
IF O2 THEN OFFSET := OFFSET + offset_2; END_IF;
IF O3 THEN OFFSET := OFFSET + offset_3; END_IF;
IF O4 THEN OFFSET := OFFSET + offset_4; END_IF;



(* revision history
hm	12. jan 2007
	original version


*)
          
END_FUNCTION

FUNCTION OFFSET2 : REAL
  VAR_INPUT
    X : REAL;
    O1 : BOOL;
    O2 : BOOL;
    O3 : BOOL;
    O4 : BOOL;
    D : BOOL;
    {attribute 'input_constant'}
    Offset_1 : REAL;
    {attribute 'input_constant'}
    Offset_2 : REAL;
    {attribute 'input_constant'}
    Offset_3 : REAL;
    {attribute 'input_constant'}
    Offset_4 : REAL;
    {attribute 'input_constant'}
    default : REAL;
  END_VAR

            IF D THEN OFFSET2 := default; ELSE OFFSET2 := X; END_IF;
IF O4 THEN OFFSET2 := OFFSET2 + offset_4;
ELSIF O3 THEN OFFSET2 := OFFSET2 + offset_3;
ELSIF O2 THEN OFFSET2 := OFFSET2 + offset_2;
ELSIF O1 THEN OFFSET2 := OFFSET2 + offset_1;
END_IF;
          
END_FUNCTION

FUNCTION OVERRIDE : REAL
  VAR_INPUT
    X1 : REAL;
    X2 : REAL;
    X3 : REAL;
    E1 : BOOL;
    E2 : BOOL;
    E3 : BOOL;
  END_VAR

            IF E1 THEN OVERRIDE := X1; END_IF;
IF E2 AND ABS(x2) > ABS(OVERRIDE) THEN OVERRIDE := X2; END_IF;
IF E3 AND ABS(x3) > ABS(OVERRIDE) THEN OVERRIDE := X3; END_IF;

(* revision history
hm	4.11.2007		rev 1.0
	original version

*)

          
END_FUNCTION

FUNCTION RANGE_TO_BYTE : BYTE
  VAR_INPUT
    X : REAL;
    low : REAL;
    high : REAL;
  END_VAR

            RANGE_TO_BYTE := INT_TO_BYTE(TRUNC_INT((LIMIT(low, X, high) - low) * 255.0 / (high - low)));


(* revision history
hm	9. jan 2008		rev 1.0
	original version

*)

          
END_FUNCTION

FUNCTION RANGE_TO_WORD : WORD
  VAR_INPUT
    X : REAL;
    low : REAL;
    high : REAL;
  END_VAR

            RANGE_TO_WORD := DINT_TO_WORD(TRUNC_INT((LIMIT(low,X,high)-low) * 65535.0 / (high - low)));


(* revision history
hm	9. jan 2008		rev 1.0
	original version

*)

          
END_FUNCTION

FUNCTION SCALE : REAL
  VAR_INPUT
    X : REAL;
    K : REAL;
    O : REAL;
    MX : REAL;
    MN : REAL;
  END_VAR

            SCALE := LIMIT(MN, X * K + O, MX);


(* revision history
hm	16. may. 2008		rev 1.0
	original version
*)
          
END_FUNCTION

FUNCTION SCALE_B : REAL
  VAR_INPUT
    X : BYTE;
    I_LO : BYTE;
    I_HI : BYTE;
    O_LO : REAL;
    O_HI : REAL;
  END_VAR

            IF I_HI = I_LO THEN
	SCALE_B := O_LO;
ELSE
	SCALE_B := (O_HI - O_LO) / BYTE_TO_REAL(I_HI - I_LO) * BYTE_TO_REAL(LIMIT(I_LO, X, I_HI));
END_IF

(* revision history
hm	18. may. 2008		rev 1.0
	original version

hm	18. jan 2011		rev 1.1
	avoid division by 0

*)
          
END_FUNCTION

FUNCTION SCALE_B2 : REAL
  VAR_INPUT
    in1 : BYTE;
    in2 : BYTE;
    K : REAL;
    O : REAL;
    {attribute 'input_constant'}
    in1_min : REAL;
    {attribute 'input_constant'}
    in1_max : REAL := 1000;
    {attribute 'input_constant'}
    in2_min : REAL;
    {attribute 'input_constant'}
    in2_max : REAL := 1000;
  END_VAR

            SCALE_B2 := 	(((in1_max - in1_min)* in1 + (in2_max - in2_min)* in2) * 0.003921569 + in1_min + in2_min) * K + O;


(* revision History
hm 19.1.2007		rev 1.1
	changed outputs to real to avoid overflow of integer
	added offset for better cascading of scale functions
	changed from FB to function

hm	6. jan 2008		rev 1.2
	improved performance

hm	26. oct. 2008	rev 1.3
	code optimization

hm	3. nov. 2008	rev 1.4
	used wrong factor in formula

*)
          
END_FUNCTION

FUNCTION SCALE_B4 : REAL
  VAR_INPUT
    in1 : BYTE;
    in2 : BYTE;
    in3 : BYTE;
    in4 : BYTE;
    K : REAL;
    O : REAL;
    {attribute 'input_constant'}
    in1_min : REAL;
    {attribute 'input_constant'}
    in1_max : REAL := 1000;
    {attribute 'input_constant'}
    in2_min : REAL;
    {attribute 'input_constant'}
    in2_max : REAL := 1000;
    {attribute 'input_constant'}
    in3_min : REAL;
    {attribute 'input_constant'}
    in3_max : REAL := 1000;
    {attribute 'input_constant'}
    in4_min : REAL;
    {attribute 'input_constant'}
    in4_max : REAL := 1000;
  END_VAR

            SCALE_B4 := 	(((in1_max - in1_min)* in1 + (in2_max - in2_min)* in2 + (in3_max - in3_min)* in3 + (in4_max - in4_min)* in4)* 0.003921569 + in1_min + in2_min + in3_min + in4_min) * K + O;


(* revision History
hm 19.1.2007		rev 1.1
	changed outputs to real to avoid overflow of integer
	added offset for better cascading of scale functions
	changed from fb to function

hm	6. jan 2008		rev 1.2
	improved performance

hm	26. oct. 2008	rev 1.3
	optimized code

hm	3. nov. 2008	rev 1.4
	used wrong factor in formula

*)
          
END_FUNCTION

FUNCTION SCALE_B8 : REAL
  VAR_INPUT
    in1 : BYTE;
    in2 : BYTE;
    in3 : BYTE;
    in4 : BYTE;
    in5 : BYTE;
    in6 : BYTE;
    in7 : BYTE;
    in8 : BYTE;
    K : REAL;
    O : REAL;
    {attribute 'input_constant'}
    in1_min : REAL;
    {attribute 'input_constant'}
    in1_max : REAL := 1000;
    {attribute 'input_constant'}
    in2_min : REAL;
    {attribute 'input_constant'}
    in2_max : REAL := 1000;
    {attribute 'input_constant'}
    in3_min : REAL;
    {attribute 'input_constant'}
    in3_max : REAL := 1000;
    {attribute 'input_constant'}
    in4_min : REAL;
    {attribute 'input_constant'}
    in4_max : REAL := 1000;
    {attribute 'input_constant'}
    in5_min : REAL;
    {attribute 'input_constant'}
    in5_max : REAL := 1000;
    {attribute 'input_constant'}
    in6_min : REAL;
    {attribute 'input_constant'}
    in6_max : REAL := 1000;
    {attribute 'input_constant'}
    in7_min : REAL;
    {attribute 'input_constant'}
    in7_max : REAL := 1000;
    {attribute 'input_constant'}
    in8_min : REAL;
    {attribute 'input_constant'}
    in8_max : REAL := 1000;
  END_VAR

            SCALE_B8 := 	(((in1_max - in1_min)* in1 + (in2_max - in2_min)* in2 + (in3_max - in3_min)* in3 + (in4_max - in4_min)* in4 +
				(in5_max - in5_min)* in5 + (in6_max - in6_min)* in6 + (in7_max - in7_min)* in7 + (in8_max - in8_min)* in8) * 0.003921569
				 + in1_min + in2_min + in3_min + in4_min + in5_min + in6_min + in7_min + in8_min) * K + O;


(* revision History
hm	19. jan.2007	rev 1.1
	changed outputs to real to avoid overflow of integer
	added offset for better cascading of scale functions

hm	6. jan. 2008	rev 1.2
	improved performance

hm	26. oct. 2008	rev 1.3
	code optimization

hm	3. nov. 2008	rev 1.4
	used wrong factor in formula

*)
          
END_FUNCTION

FUNCTION SCALE_D : REAL
  VAR_INPUT
    X : DWORD;
    I_LO : DWORD;
    I_HI : DWORD;
    O_LO : REAL;
    O_HI : REAL;
  END_VAR

            IF I_HI = I_LO THEN
	SCALE_D := O_LO;
ELSE
	SCALE_D := (O_HI - O_LO) / DWORD_TO_REAL(I_HI - I_LO) * DWORD_TO_REAL(LIMIT(I_LO, X, I_HI) - I_LO) + O_LO;
END_IF;

(* revision history
hm	18. may. 2008	rev 1.0
	original version

hm	13. nov. 2008	rev 1.1
	corrected formula for negative gradient

hm	11. jan 2011	rev 1.2
	avoid division by 0
*)
          
END_FUNCTION

FUNCTION SCALE_R : REAL
  VAR_INPUT
    X : REAL;
    I_LO : REAL;
    I_HI : REAL;
    O_LO : REAL;
    O_HI : REAL;
  END_VAR

            IF I_LO = I_HI THEN
	SCALE_R := O_LO;
ELSE
	SCALE_R := (O_HI - O_LO) / (I_HI - I_LO) * (LIMIT(I_LO, X, I_HI) - I_LO) + O_LO;
END_IF;


(* revision history
hm	18. may. 2008	rev 1.0
	original version

hm	13. nov. 2008	rev 1.1
	corrected formula for negative gradient

hm	11. jan 2011	rev 1.2
	avoid division by 0

*)
          
END_FUNCTION

FUNCTION SCALE_X2 : REAL
  VAR_INPUT
    IN1 : BOOL;
    IN2 : BOOL;
    K : REAL;
    O : REAL;
    {attribute 'input_constant'}
    IN1_MIN : REAL;
    {attribute 'input_constant'}
    IN1_MAX : REAL := 1000;
    {attribute 'input_constant'}
    IN2_MIN : REAL;
    {attribute 'input_constant'}
    IN2_MAX : REAL := 1000;
  END_VAR

            SCALE_X2 := (SEL(IN1, IN1_MIN, IN1_MAX)+ SEL(IN2, IN2_MIN, IN2_MAX)) * k + o;


(* revision history
hm	19. jan, 2007	rev 1.0
	original version

hm	26. oct. 2008	rev 1.1
	code optimized

*)
          
END_FUNCTION

FUNCTION SCALE_X4 : REAL
  VAR_INPUT
    IN1 : BOOL;
    IN2 : BOOL;
    IN3 : BOOL;
    IN4 : BOOL;
    K : REAL;
    O : REAL;
    {attribute 'input_constant'}
    IN1_MIN : REAL;
    {attribute 'input_constant'}
    IN1_MAX : REAL := 1000;
    {attribute 'input_constant'}
    IN2_MIN : REAL;
    {attribute 'input_constant'}
    IN2_MAX : REAL := 1000;
    {attribute 'input_constant'}
    IN3_MIN : REAL;
    {attribute 'input_constant'}
    IN3_MAX : REAL := 1000;
    {attribute 'input_constant'}
    IN4_MIN : REAL;
    {attribute 'input_constant'}
    IN4_MAX : REAL := 1000;
  END_VAR

            SCALE_X4 := (SEL(IN1,IN1_MIN, IN1_MAX) + SEL(IN2, IN2_MIN, IN2_MAX)+SEL(IN3, IN3_MIN, IN3_MAX)+ SEL(IN4, IN4_MIN, IN4_MAX)) * k + o;


(* revision history
hm	19. jan. 2008	rev 1.0
	original version

hm	26. oct. 2008	rev 1.1
	optimized code
*)
          
END_FUNCTION

FUNCTION SCALE_X8 : REAL
  VAR_INPUT
    in1 : BOOL;
    in2 : BOOL;
    in3 : BOOL;
    in4 : BOOL;
    in5 : BOOL;
    in6 : BOOL;
    in7 : BOOL;
    in8 : BOOL;
    K : REAL;
    O : REAL;
    {attribute 'input_constant'}
    in1_min : REAL;
    {attribute 'input_constant'}
    in1_max : REAL := 1000;
    {attribute 'input_constant'}
    in2_min : REAL;
    {attribute 'input_constant'}
    in2_max : REAL := 1000;
    {attribute 'input_constant'}
    in3_min : REAL;
    {attribute 'input_constant'}
    in3_max : REAL := 1000;
    {attribute 'input_constant'}
    in4_min : REAL;
    {attribute 'input_constant'}
    in4_max : REAL := 1000;
    {attribute 'input_constant'}
    in5_min : REAL;
    {attribute 'input_constant'}
    in5_max : REAL := 1000;
    {attribute 'input_constant'}
    in6_min : REAL;
    {attribute 'input_constant'}
    in6_max : REAL := 1000;
    {attribute 'input_constant'}
    in7_min : REAL;
    {attribute 'input_constant'}
    in7_max : REAL := 1000;
    {attribute 'input_constant'}
    in8_min : REAL;
    {attribute 'input_constant'}
    in8_max : REAL := 1000;
  END_VAR

            SCALE_X8 := (SEL(IN1,IN1_MIN, IN1_MAX)+ SEL(IN2,IN2_MIN, IN2_MAX)+SEL(IN3,IN3_MIN, IN3_MAX)+ SEL(IN4,IN4_MIN, IN4_MAX)
				+SEL(IN5,IN5_MIN, IN5_MAX)+ SEL(IN6,IN6_MIN, IN6_MAX)+SEL(IN7,IN7_MIN, IN7_MAX)+ SEL(IN8,IN8_MIN, IN8_MAX)) * k + o;



(* revision history
hm	19. jan. 2008	rev 1.0
	original version

hm	26. oct. 2008	rev 1.1
	optimized code

hm	24. jan. 2008	rev 1.2
	corrected error in formula
*)
          
END_FUNCTION

FUNCTION_BLOCK SEL2_OF_3
  VAR_INPUT
    IN1 : REAL;
    IN2 : REAL;
    IN3 : REAL;
    D : REAL;
  END_VAR
  VAR_OUTPUT
    Y : REAL;
    W : INT;
    E : BOOL;
  END_VAR
  VAR
    D12 : BOOL;
    D23 : BOOL;
    D31 : BOOL;
  END_VAR

            D12 := ABS(IN1-IN2) <= D;
D23 := ABS(IN2-IN3) <= D;
D31 := ABS(IN3-IN1) <= D;

IF (D12 AND D23) OR (D12 AND D31) OR (D23 AND D31) THEN
	(* all 3 inputs are valid *)
	Y := (IN1 + IN2 + IN3) * 0.333333333333;
	E := FALSE;
	W := 0;
ELSIF D12 THEN
	(* only inut 1 and 2 are valid *)
	Y := (In1 + IN2) * 0.5;
	E := FALSE;
	W := 3;
ELSIF D23 THEN
	(* only inut 2 and 3 are valid *)
	Y := (In2 + IN3) * 0.5;
	E := FALSE;
	W := 1;
ELSIF D31 THEN
	(* only inut 3 and 1 are valid *)
	Y := (In3 + IN1) * 0.5;
	E := FALSE;
	W := 2;
ELSE
	(* no calculation possible *)
	E := TRUE;
	W := 4;
END_IF;


(* revision history
hm	18. may 2008	rev 1.0
	original version

hm	10. mar. 2009	rev 1.1
	improved code
*)
          
END_FUNCTION_BLOCK

FUNCTION_BLOCK SEL2_OF_3B
  VAR_INPUT
    IN1 : BOOL;
    IN2 : BOOL;
    IN3 : BOOL;
    TD : TIME;
  END_VAR
  VAR_OUTPUT
    Q : BOOL;
    W : BOOL;
  END_VAR
  VAR
    TDEL : TON;
  END_VAR

            Q := (IN1 AND IN2) OR (IN1 AND IN3) OR (IN2 AND IN3);
TDEL(IN := (in1 XOR in2) OR (in1 XOR in3) OR (in2 XOR in3), PT := TD);
W := TDEL.Q;


(* revision history
hm		19. may 2008	rev 1.0
	original version

*)
          
END_FUNCTION_BLOCK

FUNCTION_BLOCK SH
  VAR_INPUT
    in : REAL;
    CLK : BOOL;
  END_VAR
  VAR_OUTPUT
    out : REAL;
    trig : BOOL;
  END_VAR
  VAR
    edge : BOOL;
  END_VAR

            IF clk AND NOT edge THEN
	out := in;
	trig := TRUE;
ELSE;
	trig := FALSE;
END_IF;
edge := clk;

(* revision history

hm 16.1.2007	rev 1.1
	added trig output

*)
          
END_FUNCTION_BLOCK

FUNCTION_BLOCK SH_1
  VAR_INPUT
    in : REAL;
    PT : TIME;
  END_VAR
  VAR_OUTPUT
    out : REAL;
    Trig : BOOL;
  END_VAR
  VAR
    last : TIME;
    tx : TIME;
  END_VAR

            (* read system time *)
tx := DWORD_TO_TIME(T_PLC_MS());

IF tx - last >= PT THEN
	last := tx;
	out := in;
	trig := TRUE;
ELSE
	trig := FALSE;
END_IF;

(* revision history

HM	6.1.2007	rev 1.1
	added trig output

HM	17.9.2007	rev 1.2
	replaced time() with T_PLC_MS() for compatibility reasons
*)


          
END_FUNCTION_BLOCK

FUNCTION_BLOCK SH_2
  VAR_INPUT
    in : REAL;
    PT : TIME;
    N : INT := 16;
    disc : INT;
  END_VAR
  VAR_OUTPUT
    out : REAL;
    trig : BOOL;
    avg : REAL;
    high : REAL;
    low : REAL;
  END_VAR
  VAR
    M : INT;
    buf : ARRAY[0..15] OF REAL;
    buf2 : ARRAY[0..15] OF REAL;
    last : TIME;
    i : INT;
    start : INT;
    temp : REAL;
    stop : INT;
    tx : TIME;
    d2 : INT;
  END_VAR

            (* read system time *)
tx := DWORD_TO_TIME(T_PLC_MS());
d2 := SHR(disc,1);

IF tx - last >= PT THEN
	last := tx;
	trig := TRUE;

	(* limit M to 0..16 *)
	M := LIMIT(1,N,16);

	(* edge detected lets take the sample *)
	FOR i := M - 1 TO 1 BY -1 DO buf2[i] := buf2[i-1]; END_FOR;
	buf2[0] := in;
	out := in;
	buf := buf2;

	(* sort the ARRAY lowest value AT 0 *)
	FOR start := 0 TO M - 2 DO
		FOR i := start+1 TO M - 1 DO
			IF buf[start] > buf[i] THEN
				temp := buf[start];
				buf[start] := buf[i];
				buf[i] := temp;
			END_IF;
		END_FOR;
	END_FOR;

	(* any calculation with the samples is here *)
	stop := M - 1 - d2;
	start := d2;
	IF NOT even(disc) THEN start := start + 1; END_IF;
	avg := 0;
	FOR i := start TO stop DO avg := avg + buf[i]; END_FOR;
	avg := avg / INT_TO_REAL(stop - start +1);
	low := buf[start];
	high := buf[stop];
ELSE
	Trig := FALSE;
END_IF;

(* revision history
hm 20. jan. 2007	rev 1.1
	added input N to specify the amout of samples for average and high low calculations
	added trig output

hm 10. sep. 2007 	rev 1.2
	an error would be generated if N was set to 0, now n is forced to1 if set to 0.
	index was out of array.

hm	17. sep. 2007	rev 1.3
	replaced time() with t_plc_ms() for compatibility reasons

hm	6. jan. 2008	rev 1.4
	improved performance

hm	14. jun. 2008	rev 1.5
	set default for input N = 16

hm	10. mar. 2009	rev 1.6
	added type conversion for compatibility reasons

*)
          
END_FUNCTION_BLOCK

FUNCTION_BLOCK SH_T
  VAR_INPUT
    IN : REAL;
    E : BOOL;
  END_VAR
  VAR_OUTPUT
    OUT : REAL;
  END_VAR

            IF E THEN out := in; END_IF;



(* revision history
hm	1. sep. 2006	rev 1.0
	original version

hm	18. oct. 2008	rev 1.1
	changed input en to e for compatibility reasons

*)
          
END_FUNCTION_BLOCK

FUNCTION STAIR : REAL
  VAR_INPUT
    X : REAL;
    D : REAL;
  END_VAR

            IF D > 0.0 THEN
	STAIR := DINT_TO_REAL(REAL_TO_DINT(X / D)) * D;
ELSE
	STAIR := X;
END_IF;



(* revision history
hm	28 jan 2007		rev 1.0
	original version

hm	27 dec 2007		rev 1.1
	changed code for better performance

hm	6. jan 2008		rev 1.2
	further performance improvement

hm	26. oct. 2008		rev 1.3
	optimized code

hm	10. mar. 2009	rev 1.4
	real constants updated to new systax using dot

*)
          
END_FUNCTION

FUNCTION_BLOCK STAIR2
  VAR_INPUT
    X : REAL;
    D : REAL;
  END_VAR
  VAR_OUTPUT
    Y : REAL;
  END_VAR

            IF D > 0.0 THEN
	IF X >= Y + D OR X <= Y - D THEN Y := FLOOR(X/D) * D; END_IF;
ELSE
	Y := X;
END_IF;



(* revision history
hm	28 jan 2007		rev 1.0
	original version

hm	27. dec 2007	rev 1.1
	changed code for better performance

hm	30. jun. 2008	rev 1.2
	added type conversions to avoid warnings under codesys 3.0																																																																																																																																																																																																																																																											

ks	26. oct. 2008	rev 1.3
	improved code

hm	10. mar. 2009	rev 1.4
	real constants updated to new systax using dot

*)
          
END_FUNCTION_BLOCK

FUNCTION_BLOCK TREND
  VAR_INPUT
    X : REAL;
  END_VAR
  VAR_OUTPUT
    Q : BOOL;
    TU : BOOL;
    TD : BOOL;
    D : REAL;
  END_VAR
  VAR
    last_X : REAL;
  END_VAR

            TU := X > last_X;
TD := X < last_X;
Q := TU OR TD;
D := X - LAST_X;

last_X := X;



(* revision history
hm	21. aug. 2009	rev 1.0
	original version

*)

          
END_FUNCTION_BLOCK

FUNCTION_BLOCK TREND_DW
  VAR_INPUT
    X : DWORD;
  END_VAR
  VAR_OUTPUT
    Q : BOOL;
    TU : BOOL;
    TD : BOOL;
    D : DWORD;
  END_VAR
  VAR
    last_X : DWORD;
  END_VAR

            IF X > last_X THEN
	TU := TRUE;
	TD := FALSE;
	D := X - last_X;
	Q := TRUE;
ELSIF X < last_X THEN
	TD := TRUE;
	TU := FALSE;
	D := last_X - X;
	Q := FALSE;
ELSE
	TU := FALSE;
	TD := FALSE;
	D := 0;
END_IF;
last_X := X;



(* revision history
hm	21. nov. 2008	rev 1.0
	original version

hm	20. feb. 2009	rev 1.1
	added outputs TU, TD and D

hm	14. mar. 2009	rev 1.2
	removed double assignments

*)

          
END_FUNCTION_BLOCK

FUNCTION WORD_TO_RANGE : REAL
  VAR_INPUT
    X : WORD;
    low : REAL;
    high : REAL;
  END_VAR

            WORD_TO_RANGE := (high - low) * WORD_TO_REAL(X) * 0.00001525902189669640 + low;


(* revision history
hm	9. jan 2008	rev 1.0
	original version

hm	10. mar. 2009	rev 1.1
	improved code
*)

          
END_FUNCTION

FUNCTION LIST_CLEAN : BOOL
  VAR_INPUT
    SEP : BYTE;
  END_VAR
  VAR
    pt : POINTER TO ARRAY[1..LIST_LENGTH] OF BYTE;
    pos : INT;
    pw : INT;
    last : BYTE;
    c : BYTE;
  END_VAR
  VAR_IN_OUT
    LIST : STRING(LIST_LENGTH);
  END_VAR

            pt := ADR(LIST);

last := sep;
REPEAT
   pos := pos + 1;
   c := pt^[pos];
   IF last <> sep OR c <> sep THEN
      pw := pw + 1;
      pt^[pw] := c;
   END_IF;
   last := c;
UNTIL pos >= LIST_LENGTH OR c = 0
END_REPEAT;

IF pw > 1 THEN
  pw := pw - 1;
  IF pt^[pw] = sep THEN pt^[pw] := 0; END_IF;
END_IF;

(* retrun TRUE *)
LIST_CLEAN := TRUE;



(* revision histroy
hm	28. jun. 2008	rev 1.0
	original release

hm	19. jan. 2011	rev 1.1
	changed string(255) to string(LIST_LENGTH)

*)	

          
END_FUNCTION

FUNCTION LIST_GET : STRING(LIST_LENGTH)
  VAR_INPUT
    SEP : BYTE;
    POS : INT;
  END_VAR
  VAR
    i : INT := 1;
    o : INT := 1;
    pt : POINTER TO ARRAY[1..LIST_LENGTH] OF BYTE;
    po : POINTER TO ARRAY[1..LIST_LENGTH] OF BYTE;
    cnt : INT;
    c : BYTE;
  END_VAR
  VAR_IN_OUT
    LIST : STRING(LIST_LENGTH);
  END_VAR

            (* load pointers *)
pt := ADR(LIST);
po := ADR(LIST_GET);

(* search for the n-th occurence of a separation character and store position in i *)
WHILE (cnt < pos) AND (i < LIST_LENGTH) AND (pt^[i] > 0) DO
	IF pt^[i] = sep THEN cnt := cnt + 1; END_IF;
	i := i + 1;
END_WHILE;

(* copy the list element to output *)
IF i < LIST_LENGTH THEN c := pt^[i]; END_IF;
WHILE (c <> sep) AND (c > 0) AND (o < LIST_LENGTH) AND (i < LIST_LENGTH) DO
	po^[o] :=pt^[i];
	o := o + 1;
	i := i + 1;
	c := pt^[i];
END_WHILE;

(* terminate the output string *)
po^[o] := 0;



(* revision histroy
hm	20. jun. 2008	rev 1.0
	original release

hm	19. jan. 2011	rev 1.1
	changed string(255) to strring(LIST_LENGTH)

*)	

          
END_FUNCTION

FUNCTION LIST_INSERT : BOOL
  VAR_INPUT
    SEP : BYTE;
    POS : INT;
    INS : STRING(LIST_LENGTH);
  END_VAR
  VAR
    i : INT;
    pt : POINTER TO ARRAY[1..LIST_LENGTH] OF BYTE;
    cnt : INT;
    c : BYTE;
    tmp : STRING(LIST_LENGTH);
  END_VAR
  VAR_IN_OUT
    LIST : STRING(LIST_LENGTH);
  END_VAR

            (* load pointers *)
pt := ADR(LIST);

(* search for the n-th occurence of a separation character and store position in i *)
c := pt^[1];
WHILE (cnt < pos) AND (i < LIST_LENGTH) AND (c > 0) DO
	i := i + 1;
	c := pt^[i];
	IF c = sep THEN cnt := cnt + 1; END_IF;
END_WHILE;

(* copy the new element into the list *)
tmp := CHR_TO_STRING(SEP);
IF i = 0 THEN
	tmp := CONCAT(INS,tmp);
	LIST := INSERT(LIST, tmp, 0);
ELSE
	tmp := CONCAT(tmp, INS);
	LIST := INSERT(LIST, tmp, i - 1);
END_IF;


LIST_INSERT := TRUE;



(* revision histroy
hm	28. jun. 2008	rev 1.0
	original release

hm	17. dec. 2008	rev 1.1
	changes name of function chr to chr_to_string

hm	19. jan. 2011	rev 1.2
	changed string(255) to string(LIST_LENGTH)

*)	

          
END_FUNCTION

FUNCTION LIST_LEN : INT
  VAR_INPUT
    SEP : BYTE;
  END_VAR
  VAR
    pt : POINTER TO ARRAY[1..LIST_LENGTH] OF BYTE;
    l : INT;
    pos : INT;
  END_VAR
  VAR_IN_OUT
    LIST : STRING(LIST_LENGTH);
  END_VAR

            PT := ADR(LIST);
LIST_LEN := 1;
l := LEN(list);
FOR pos := 1 TO l DO
	IF pt^[pos] = SEP THEN LIST_LEN := LIST_LEN + 1; END_IF;
END_FOR;



(* code before rev 1.1
LIST_LEN := COUNT_CHAR(LIST, SEP) + 1;
*)


(* revision histroy
hm	25. jun. 2008	rev 1.0
	original release

hm	16. oct. 2008	rev 1.1
	fixed a problem where list_len would only work up to LIST_LENGTH

hm	19. jan. 2001	rev 1.2
	changed string(255) to string(LIST_LENGTH)

*)	

          
END_FUNCTION

FUNCTION_BLOCK LIST_NEXT
  VAR_INPUT
    SEP : BYTE;
    RST : BOOL;
  END_VAR
  VAR_IN_OUT
    LIST : STRING(LIST_LENGTH);
  END_VAR
  VAR_OUTPUT
    LEL : STRING(LIST_LENGTH);
    NUL : BOOL;
  END_VAR
  VAR
    pt : POINTER TO ARRAY[1..LIST_LENGTH] OF BYTE;
    stop : INT;
    start : INT;
    pos : INT := 1;
  END_VAR

            (* load pointers *)
pt := ADR(LIST);
stop := LEN(LIST);

IF rst THEN
	start := 0;
	pos := 1;
	NUL := FALSE;
END_IF;

(* search next occurence of separation character or end of list *)
WHILE pos <= stop DO
	IF pt^[pos] = SEP THEN EXIT; END_IF;
	pos := pos + 1;
END_WHILE;
IF start <= stop THEN
	LEL := MID(LIST, pos - start - 1, start + 1);
	start := pos;
	pos := pos + 1;
ELSE
	LEL := '';
	NUL := TRUE;
END_IF;



(* revision histroy
hm	25. jun. 2008	rev 1.0
	original release

hm	19. jan. 2011	rev 1.1
	changed string(255) to string(LIST_LENGTH)	

*)	

          
END_FUNCTION_BLOCK

FUNCTION LIST_RETRIEVE : STRING(LIST_LENGTH)
  VAR_INPUT
    SEP : BYTE;
    POS : INT;
  END_VAR
  VAR
    i : INT;
    o : INT;
    pt : POINTER TO ARRAY[0..LIST_LENGTH] OF BYTE;
    po : POINTER TO ARRAY[0..LIST_LENGTH] OF BYTE;
    cnt : INT;
    c : BYTE;
    p : INT;
    l : INT;
  END_VAR
  VAR_IN_OUT
    LIST : STRING(LIST_LENGTH);
  END_VAR

            (* load pointers *)
pt := ADR(LIST);
po := ADR(LIST_RETRIEVE);
l := LEN(LIST);

(* search for the n-th occurence of a separation character and store position in i *)
WHILE (cnt < pos) AND (i < LIST_LENGTH) AND (pt^[i] > 0) DO
	IF pt^[i] = sep THEN cnt := cnt + 1; END_IF;
	i := i + 1;
END_WHILE;

p := i;	(* store position for deletion in list *)

(* copy the list element to output *)
IF i < LIST_LENGTH THEN c := pt^[i]; END_IF;
WHILE (c <> sep) AND (c > 0) AND (o < LIST_LENGTH) AND (i < LIST_LENGTH) DO
	po^[o] :=pt^[i];
	o := o + 1;
	i := i + 1;
	c := pt^[i];
END_WHILE;

IF cnt = pos THEN
	IF i = L THEN
		LIST := LEFT(LIST, p - 1);
	ELSE
		LIST := DELETE(LIST, i - p + 1, p + 1);
	END_IF;
END_IF;


(* terminate the output string *)
po^[o] := 0;



(* revision histroy
hm	28. jun. 2008	rev 1.0
	original release

hm	19. jan. 2011	rev 1.1
	changed string(255) to string(LIST_LENGTH)

*)	

          
END_FUNCTION

FUNCTION LIST_RETRIEVE_MAX : STRING(LIST_LENGTH)
  VAR_INPUT
    SEP : BYTE;
  END_VAR
  VAR
    pt : POINTER TO ARRAY[1..LIST_LENGTH] OF BYTE;
    l : INT;
    pos : INT;
    last : INT;
    lx : INT;
    mpos : INT := 1;
  END_VAR
  VAR_IN_OUT
    LIST : STRING(LIST_LENGTH);
  END_VAR

            PT := ADR(LIST);
l := LEN(list);
FOR pos := 1 TO l DO
	IF pt^[pos] = sep THEN
		IF pos - last - 1 > lx THEN
			mpos := last + 1;
			lx := pos - last - 1;
		END_IF;
		last := pos;
	END_IF;
END_FOR;

(* check length of last element *)
IF l - last > lx THEN
	mpos := last + 1;
	lx := l - last;
	LIST_RETRIEVE_MAX := RIGHT(list, lx);
	list := LEFT(list, last - 1);
ELSE
	LIST_RETRIEVE_MAX := MID(LIST, lx, mpos);
	LIST := DELETE(LIST, lx + 1, mpos);
END_IF;



(* revision histroy
hm	22. oct. 2008	rev 1.0
	original release

hm	19. jan. 2011	rev 1.1
	changed string(255) to string(LIST_LENGTH)

*)	

          
END_FUNCTION

FUNCTION LIST_RETRIEVE_MIN : STRING(LIST_LENGTH)
  VAR_INPUT
    SEP : BYTE;
  END_VAR
  VAR
    pt : POINTER TO ARRAY[1..LIST_LENGTH] OF BYTE;
    l : INT;
    pos : INT;
    last : INT;
    lx : INT;
    mpos : INT := 1;
  END_VAR
  VAR_IN_OUT
    LIST : STRING(LIST_LENGTH);
  END_VAR

            PT := ADR(LIST);
l := LEN(list);
lx := 255;
FOR pos := 1 TO l DO
	IF pt^[pos] = sep THEN
		IF pos - last - 1 < lx THEN
			mpos := last + 1;
			lx := pos - last - 1;
			(* if we found an element with length 0 then we can stop *)
		END_IF;
		last := pos;
		IF lx = 0 THEN EXIT; END_IF;
	END_IF;
END_FOR;

(* check length of last element *)
IF l - last < lx THEN
	mpos := last + 1;
	lx := l - last;
	LIST_RETRIEVE_MIN := RIGHT(list, lx);
	list := LEFT(list, last - 1);
ELSE
	LIST_RETRIEVE_MIN := MID(LIST, lx, mpos);
	LIST := DELETE(LIST, lx + 1, mpos);
END_IF;



(* revision histroy
hm	23. oct. 2008	rev 1.0
	original release

hm	19. jan. 2011	rev 1.1
	changed string(255) to string(LIST_LENGTH)

*)	

          
END_FUNCTION

FUNCTION LIST_SORT_L : STRING(LIST_LENGTH)
  VAR_INPUT
    SEP : BYTE;
  END_VAR
  VAR
    element : STRING(LIST_LENGTH);
    sepx : STRING(1);
  END_VAR
  VAR_IN_OUT
    LIST : STRING(LIST_LENGTH);
  END_VAR

            sepx := CHR_TO_STRING(sep);
WHILE list <> '' DO
	IF list = sepx THEN
		LIST_SORT_L := CONCAT(sepx, LIST_SORT_L);
		list := '';
		RETURN;
	ELSE
		element := LIST_RETRIEVE_MIN(SEP,LIST);
		LIST_SORT_L := CONCAT(LIST_SORT_L, element);
		LIST_SORT_L := CONCAT(LIST_SORT_L, sepx);
	END_IF;
END_WHILE;
(* delete the last separation character *)
LIST_SORT_L := LEFT(LIST_SORT_L, LEN(LIST_SORT_L) - 1);


(* revision histroy
hm	23. oct. 2008	rev 1.0
	original release

hm	17. dec. 2008	rev 1.1
	changes name of function chr to chr_to_string

hm	19. jan. 2011	rev 1.2
	changed string(255) to string(LIST_LENGTH)

*)	

          
END_FUNCTION

FUNCTION_BLOCK COUNT_BR
  VAR_INPUT
    SET : BOOL;
    IN : BYTE;
    UP : BOOL;
    DN : BOOL;
    STEP : BYTE := 1;
    MX : BYTE := 255;
    RST : BOOL;
  END_VAR
  VAR_OUTPUT
    CNT : BYTE;
  END_VAR
  VAR
    last_up : BOOL;
    last_dn : BOOL;
  END_VAR

            IF rst THEN
	cnt := 0;
ELSIF set THEN
	cnt := LIMIT(0,in,mx);
ELSIF up AND NOT last_up THEN
	cnt := INT_TO_BYTE(INC(cnt,step,mx));
ELSIF dn AND NOT last_dn THEN
	cnt := INT_TO_BYTE(inc(cnt,-step,mx));
END_IF;
last_up := up;
last_dn := dn;

(* revision history
hm	16. jan 2008	rev 1.0
	original version

*)
          
END_FUNCTION_BLOCK

FUNCTION_BLOCK COUNT_DR
  VAR_INPUT
    SET : BOOL;
    IN : DWORD;
    UP : BOOL;
    DN : BOOL;
    STEP : DWORD := 1;
    MX : DWORD := 16#FFFFFFFF;
    RST : BOOL;
  END_VAR
  VAR_OUTPUT
    CNT : DWORD;
  END_VAR
  VAR
    last_up : BOOL;
    last_dn : BOOL;
  END_VAR

            IF rst THEN
	cnt := 0;
ELSIF set THEN
	cnt := LIMIT(0,in,mx);
ELSIF up AND NOT last_up THEN
	IF STEP > MX - CNT THEN
		CNT := CNT - MX + STEP - 1;
	ELSE
		CNT := CNT + STEP;
	END_IF;
ELSIF dn AND NOT last_dn THEN
	IF STEP > CNT THEN
		CNT := CNT - STEP + MX + 1;
	ELSE
		CNT := CNT - STEP;
	END_IF;
END_IF;
last_up := up;
last_dn := dn;

(* revision history
hm	12. jun 2008	rev 1.0
	original version

hm	20. jan. 2011	rev 1.1
	corrected init value of MX to 16#FFFFFFFF

*)
          
END_FUNCTION_BLOCK

FUNCTION_BLOCK FF_D2E
  VAR_INPUT
    D0 : BOOL;
    D1 : BOOL;
    CLK : BOOL;
    RST : BOOL;
  END_VAR
  VAR_OUTPUT
    Q0 : BOOL;
    Q1 : BOOL;
  END_VAR
  VAR
    edge : BOOL;
  END_VAR

            IF rst THEN
	Q0 := FALSE;
	Q1 := FALSE;
ELSIF clk AND NOT edge THEN
	Q0 := D0;
	Q1 := D1;
END_IF;
edge := CLK;

(* revision history
hm	25. dec 2007	rev 1.0
	original version

hm	27. dec 2007	rev 1.1
	changed code for better performance

hm	30. oct. 200	rev 1.2
	deleted unnecessary init with 0

hm	14. mar. 2009	rev 1.3
	removed double assignments

*)

          
END_FUNCTION_BLOCK

FUNCTION_BLOCK FF_D4E
  VAR_INPUT
    D0 : BOOL;
    D1 : BOOL;
    D2 : BOOL;
    D3 : BOOL;
    CLK : BOOL;
    RST : BOOL;
  END_VAR
  VAR_OUTPUT
    Q0 : BOOL;
    Q1 : BOOL;
    Q2 : BOOL;
    Q3 : BOOL;
  END_VAR
  VAR
    edge : BOOL;
  END_VAR

            IF rst THEN
	Q0 := FALSE;
	Q1 := FALSE;
	Q2 := FALSE;
	Q3 := FALSE;
ELSIF clk AND NOT edge THEN
	Q0 := D0;
	Q1 := D1;
	Q2 := D2;
	Q3 := D3;
END_IF;
edge := CLK;

(* revision history
hm	4. aug 2006	rev 1.0
	original version

hm	27. dec 2007	rev 1.1
	changed code for better performance

hm	30. oct. 200	rev 1.2
	deleted unnecessary init with 0

hm	14. mar. 2009	rev 1.3
	removed double assignments

*)

          
END_FUNCTION_BLOCK

FUNCTION_BLOCK FF_DRE
  VAR_INPUT
    SET : BOOL;
    D : BOOL;
    CLK : BOOL;
    RST : BOOL;
  END_VAR
  VAR_OUTPUT
    Q : BOOL;
  END_VAR
  VAR
    edge : BOOL;
  END_VAR

            IF rst OR set THEN
	Q := NOT rst;
ELSIF clk AND NOT edge THEN
	Q := D;
END_IF;
edge := CLK;

(* revision history
hm	4. aug 2006		rev 1.0
	original version

hm	27. dec 2007	rev 1.1
	changed code for better performance

hm	30. oct. 2008	rev 1.2
	optimized performance
*)
          
END_FUNCTION_BLOCK

FUNCTION_BLOCK FF_JKE
  VAR_INPUT
    SET : BOOL;
    J : BOOL;
    CLK : BOOL;
    K : BOOL;
    RST : BOOL;
  END_VAR
  VAR_OUTPUT
    Q : BOOL;
  END_VAR
  VAR
    edge : BOOL;
  END_VAR

            IF rst OR set THEN
	Q := NOT rst;
ELSIF clk AND NOT edge THEN
	IF J XOR K THEN Q := J;
	ELSE Q := K XOR Q;
	END_IF;
END_IF;
edge := CLK;

(* revision history
hm	4. aug 2006		rev 1.0
	original version

hm	27. dec 2007	rev 1.1
	changed code for better performance

hm	30. oct. 2008	rev 1.2
	optimized performance
*)
          
END_FUNCTION_BLOCK

FUNCTION_BLOCK FF_RSE
  VAR_INPUT
    CS : BOOL;
    CR : BOOL;
    RST : BOOL;
  END_VAR
  VAR_OUTPUT
    Q : BOOL;
  END_VAR
  VAR
    es : BOOL;
    er : BOOL;
  END_VAR

            IF rst THEN
	(* asynchronous reset *)
	Q := FALSE;
ELSIF CR AND NOT er THEN
	(* rising edge on CR *)
	Q := FALSE;
ELSIF CS AND NOT es THEN
	(* rising edge on CS *)
	Q := TRUE;
END_IF;

es := CS;
er := CR;

(* revision history

hm	16. jul. 2008	rev 1.0
	original version

*)




          
END_FUNCTION_BLOCK

FUNCTION_BLOCK SELECT_8
  VAR_INPUT
    E : BOOL;
    SET : BOOL;
    IN : BYTE;
    UP : BOOL;
    DN : BOOL;
    RST : BOOL;
  END_VAR
  VAR_OUTPUT
    Q0 : BOOL;
    Q1 : BOOL;
    Q2 : BOOL;
    Q3 : BOOL;
    Q4 : BOOL;
    Q5 : BOOL;
    Q6 : BOOL;
    Q7 : BOOL;
    STATE : INT;
  END_VAR
  VAR
    last_up : BOOL;
    last_dn : BOOL;
  END_VAR

            IF rst THEN
	state := 0;
ELSIF set THEN
	state := IN;
ELSIF up AND NOT last_up THEN
	state := inc(state,1,7);
ELSIF dn AND NOT last_dn THEN
	state := inc(state,-1,7);
END_IF;
last_UP := UP;
last_DN := DN;

Q0 := FALSE;
Q1 := FALSE;
Q2 := FALSE;
Q3 := FALSE;
Q4 := FALSE;
Q5 := FALSE;
Q6 := FALSE;
Q7 := FALSE;

IF E THEN
	CASE state OF
		0: Q0 := TRUE;
		1: Q1 := TRUE;
		2: Q2 := TRUE;
		3: Q3 := TRUE;
		4: Q4 := TRUE;
		5: Q5 := TRUE;
		6: Q6 := TRUE;
		7: Q7 := TRUE;
	END_CASE;
END_IF;

(* revision history
hm	16. jan 2008	rev 1.0
	original version

hm	27. feb. 2009	rev 1.1
	renamed input en to e
*)
          
END_FUNCTION_BLOCK

FUNCTION_BLOCK SHR_4E
  VAR_INPUT
    SET : BOOL;
    D0 : BOOL;
    CLK : BOOL;
    RST : BOOL;
  END_VAR
  VAR_OUTPUT
    Q0 : BOOL;
    Q1 : BOOL;
    Q2 : BOOL;
    Q3 : BOOL;
  END_VAR
  VAR
    trig : R_TRIG;
  END_VAR

            (* trig.Q signals a rising edge on clk *)
trig(clk := clk);

IF set OR rst THEN
	Q0 := NOT rst;
	Q1 := Q0;
	Q2 := Q0;
	Q3 := Q0;
ELSIF trig.Q THEN
	Q3 := Q2;
	Q2 := Q1;
	Q1 := Q0;
	Q0 := D0;
END_IF;



(* revision history
hm	4. aug. 2006	rev 1.0
	original version

hm	25. oct. 2008	rev 1.1
	optimized code

*)
          
END_FUNCTION_BLOCK

FUNCTION_BLOCK SHR_4UDE
  VAR_INPUT
    SET : BOOL;
    D0 : BOOL;
    D3 : BOOL;
    CLK : BOOL;
    DN : BOOL;
    RST : BOOL;
  END_VAR
  VAR_OUTPUT
    Q0 : BOOL;
    Q1 : BOOL;
    Q2 : BOOL;
    Q3 : BOOL;
  END_VAR
  VAR
    trig : R_TRIG;
  END_VAR

            (* trig.Q signals a rising edge on clk *)
trig(clk := clk);

IF set OR rst THEN
	Q0 := NOT RST;
	Q1 := Q0;
	Q2 := Q0;
	Q3 := Q0;
ELSIF trig.Q THEN
	IF dn THEN
		Q0 := Q1;
		Q1 := Q2;
		Q2 := Q3;
		Q3 := D3;
	ELSE
		Q3 := Q2;
		Q2 := Q1;
		Q1 := Q0;
		Q0 := D0;
	END_IF;
END_IF;



(* revision history
hm	4. aug. 2006	rev 1.0
	original version

hm	25. oct. 2008	rev 1.1
	optimized code

hm	14. mar. 2009	rev 1.2
	removed double assignments

*)
          
END_FUNCTION_BLOCK

FUNCTION_BLOCK SHR_8PLE
  VAR_INPUT
    Din : BOOL;
    Dload : BYTE;
    CLK : BOOL;
    UP : BOOL := 1;
    load : BOOL;
    RST : BOOL;
  END_VAR
  VAR_OUTPUT
    DOut : BOOL;
  END_VAR
  VAR
    edge : BOOL := 1;
    register : BYTE;
  END_VAR

            (* flankenerkennung clk wird high und edge war high reset ist nicht aktiv und set ist nicht aktiv *)
IF CLK AND edge AND NOT rst THEN
	edge := FALSE;	(* flanke wurde erkannt und weitere flankenerkennung wird verhindert bis edge wieder true ist *)
	(* hier ist der code für das flankenevent *)
	IF UP THEN						(*shift up *)
		register := SHL(register,1);
		register.0 := Din;
		Dout := register.7;
	ELSE								(* shift down *);
		register := SHR(register,1);
		register.7 := Din;
		Dout := register.0;
	END_IF;
	IF load THEN							(* the byte on Din will be loaded if load = true *)
		register := Dload;
		IF up THEN Dout := register.7; ELSE Dout := register.0; END_IF;
	END_IF;
END_IF;
IF NOT clk THEN edge := TRUE; END_IF;	(* sobald clk wieder low wird warten auf nächste flanke *)
IF rst THEN									(* wenn reset aktiv dann ausgang rücksetzen *)
	register := 0;
	Dout := FALSE;
END_IF;

          
END_FUNCTION_BLOCK

FUNCTION_BLOCK SHR_8UDE
  VAR_INPUT
    SET : BOOL;
    D0 : BOOL;
    D7 : BOOL;
    CLK : BOOL;
    DN : BOOL;
    RST : BOOL;
  END_VAR
  VAR_OUTPUT
    Q0 : BOOL;
    Q1 : BOOL;
    Q2 : BOOL;
    Q3 : BOOL;
    Q4 : BOOL;
    Q5 : BOOL;
    Q6 : BOOL;
    Q7 : BOOL;
  END_VAR
  VAR
    trig : R_TRIG;
  END_VAR

            (* trig.Q signals a rising edge on clk *)
trig(clk := clk);

IF set OR rst THEN
	Q0 := NOT RST;
	Q1 := Q0;
	Q2 := Q0;
	Q3 := Q0;
	Q4 := Q0;
	Q5 := Q0;
	Q6 := Q0;
	Q7 := Q0;
ELSIF trig.Q THEN
	IF dn THEN
		Q0 := Q1;
		Q1 := Q2;
		Q2 := Q3;
		Q3 := Q4;
		Q4 := Q5;
		Q5 := Q6;
		Q6 := Q7;
		Q7 := D7;
	ELSE
		Q7 := Q6;
		Q6 := Q5;
		Q5 := Q4;
		Q4 := Q3;
		Q3 := Q2;
		Q2 := Q1;
		Q1 := Q0;
		Q0 := D0;
	END_IF;
END_IF;



(* revision history
hm	4. aug. 2006	rev 1.0
	original version

hm	25. oct. 2008	rev 1.1
	optimized code

hm	14. mar. 2009	rev 1.2
	removed double assignments

*)
          
END_FUNCTION_BLOCK

FUNCTION_BLOCK TOGGLE
  VAR_INPUT
    CLK : BOOL;
    rst : BOOL;
  END_VAR
  VAR_OUTPUT
    Q : BOOL;
  END_VAR
  VAR
    edge : BOOL;
  END_VAR

            IF rst THEN
	q := 0;
ELSIF clk AND NOT edge THEN
	Q := NOT Q;
END_IF;
edge := clk;

(* revision history

hm	13.9.2007		rev 1.0
	original version

hm	30. oct. 2008	rev 1.1
	deleted unnecessary init

*)




          
END_FUNCTION_BLOCK

FUNCTION_BLOCK LTCH
  VAR_INPUT
    D : BOOL;
    L : BOOL;
    RST : BOOL;
  END_VAR
  VAR_OUTPUT
    Q : BOOL;
  END_VAR

            (* as long as L is true, the latch is transparent and and change of D is transferred to Q *)
(* of course only when there is no asynchronous reset *)
IF rst THEN				(* if asynchronous reset then Q=0 *)
	Q := FALSE;
ELSIF L THEN			(* latch is transparent *)
	Q := D;
END_IF;


(* revision history
hm	4. aug 2006		rev 1.0
	original version

hm	27. dec 2007	rev 1.1
	changed code for better performance

hm	30. oct. 2008	rev 1.2
	deleted unnecessary init with 0

*)
          
END_FUNCTION_BLOCK

FUNCTION_BLOCK LTCH_4
  VAR_INPUT
    D0 : BOOL;
    D1 : BOOL;
    D2 : BOOL;
    D3 : BOOL;
    L : BOOL;
    RST : BOOL;
  END_VAR
  VAR_OUTPUT
    Q0 : BOOL;
    Q1 : BOOL;
    Q2 : BOOL;
    Q3 : BOOL;
  END_VAR

            (* as long as L is true, the latch is transparent and and change of D is transferred to Q *)
(* of course only when there is no asynchronous reset *)
IF rst THEN			(* if asynchronous reset then Q=0 *)
	Q0 := FALSE;
	Q1 := FALSE;
	Q2 := FALSE;
	Q3 := FALSE;
ELSIF L THEN			(* latch is transparent *)
	Q0 := D0;
	Q1 := D1;
	Q2 := D2;
	Q3 := D3;
END_IF;

(* revision history
hm	4. aug 2006	rev 1.0
	original version

hm	27. dec 2007	rev 1.1
	changed code for better performance

hm	30. oct. 2008	rev 1.2
	deleted unnecessary init with 0

hm	14. mar. 2009	rev 1.3
	removed double assignments

*)
          
END_FUNCTION_BLOCK

FUNCTION_BLOCK STORE_8
  VAR_INPUT
    Set : BOOL;
    D0 : BOOL;
    D1 : BOOL;
    D2 : BOOL;
    D3 : BOOL;
    D4 : BOOL;
    D5 : BOOL;
    D6 : BOOL;
    D7 : BOOL;
    Clr : BOOL;
    Rst : BOOL;
  END_VAR
  VAR_OUTPUT
    Q0 : BOOL;
    Q1 : BOOL;
    Q2 : BOOL;
    Q3 : BOOL;
    Q4 : BOOL;
    Q5 : BOOL;
    Q6 : BOOL;
    Q7 : BOOL;
  END_VAR
  VAR
    edge : BOOL;
  END_VAR

            IF rst OR set THEN
	q0 := NOT rst;
	q1 := q0;
	q2 := q0;
	q3 := q0;
	q4 := q0;
	q5 := q0;
	q6 := q0;
	q7 := q0;
ELSE
	IF D0 THEN Q0 := TRUE; END_IF;
	IF D1 THEN Q1 := TRUE; END_IF;
	IF D2 THEN Q2 := TRUE; END_IF;
	IF D3 THEN Q3 := TRUE; END_IF;
	IF D4 THEN Q4 := TRUE; END_IF;
	IF D5 THEN Q5 := TRUE; END_IF;
	IF D6 THEN Q6 := TRUE; END_IF;
	IF D7 THEN Q7 := TRUE; END_IF;

	IF clr AND NOT edge THEN
		IF q0 THEN q0 := FALSE;
		ELSIF q1 THEN q1 := FALSE;
		ELSIF q2 THEN q2 := FALSE;
		ELSIF q3 THEN q3 := FALSE;
		ELSIF q4 THEN q4 := FALSE;
		ELSIF q5 THEN q5 := FALSE;
		ELSIF q6 THEN q6 := FALSE;
		ELSE q7 := FALSE;
		END_IF;
	END_IF;
	edge := clr;
END_IF;


(* revision history
hm	25.12.2007	rev 1.0
	original version

hm	30. oct. 2008	rev 1.1
	optimized performance

hm	14. mar. 2009	rev 1.2
	removed double assignments

*)


          
END_FUNCTION_BLOCK

FUNCTION BCDC_TO_INT : INT
  VAR_INPUT
    IN : BYTE;
  END_VAR

            BCDC_TO_INT := (in AND 16#0F) + (SHR(in,4) * 10);

(* revision history
hm	13.12.2007	rev 1.0
	original version

hm	30.6.2008	rev 1.1
	changed name BCD_TO_INT to BCDC_TO_INT to avoid collision with util.lib

*)
          
END_FUNCTION

FUNCTION BIT_COUNT : INT
  VAR_INPUT
    IN : DWORD;
  END_VAR

            WHILE in > 0 DO
	IF in.0 THEN Bit_Count := Bit_Count + 1; END_IF;
	in := SHR(in,1);
END_WHILE;



(* revision history
5.7.2007	rev 1.0		original version

10.9.2007	rev 1.1		hm
	changed algorithm for better performace
	the execution time has reduced by a factor of 5
	deleted unused variable temp
*)
          
END_FUNCTION

FUNCTION BIT_LOAD_B : BYTE
  VAR_INPUT
    IN : BYTE;
    VAL : BOOL;
    POS : INT;
  END_VAR
  VAR CONSTANT
    dat : BYTE := 1;
  END_VAR

            IF VAL THEN
	BIT_LOAD_B := in OR SHL(dat,pos);
ELSE
	BIT_LOAD_B := in AND (NOT SHL(dat,pos));
END_IF;


(* revision history
hm	29. feb 2008	rev 1.0
	original version

hm	16. mar 2008	rev 1.1
	change input bit to val for compatibility reasons
*)

          
END_FUNCTION

FUNCTION BIT_LOAD_B2 : BYTE
  VAR_INPUT
    I : BYTE;
    D : BOOL;
    P : INT;
    N : INT;
  END_VAR

            IF D THEN
	BIT_LOAD_B2 := ROL(SHR(BYTE#255, 8 - N) OR ROR(i, P), P);
ELSE
	BIT_LOAD_B2 := ROL(SHL(BYTE#255, N) AND ROR(I, P), P);
END_IF;



(* revision history
hm	18. oct. 2008	rev 1.0
	original version


*)

          
END_FUNCTION

FUNCTION BIT_LOAD_DW : DWORD
  VAR_INPUT
    IN : DWORD;
    VAL : BOOL;
    POS : INT;
  END_VAR
  VAR CONSTANT
    dat : DWORD := 1;
  END_VAR

            IF val THEN
	BIT_LOAD_DW := in OR SHL(dat,pos);
ELSE
	BIT_LOAD_DW := in AND (NOT SHL(dat,pos));
END_IF;


(* revision history
hm	29. feb 2008	rev 1.0
	original version

hm	16. mar 2008	rev 1.1
	change input bit to val for compatibility reasons
*)


          
END_FUNCTION

FUNCTION BIT_LOAD_DW2 : DWORD
  VAR_INPUT
    I : DWORD;
    D : BOOL;
    P : INT;
    N : INT;
  END_VAR

            IF D THEN
	BIT_LOAD_DW2 := ROL(SHR(DWORD#4294967295, 32 - N) OR ROR(i, P), P);
ELSE
	BIT_LOAD_DW2 := ROL(SHL(DWORD#4294967295, N) AND ROR(I, P), P);
END_IF;



(* revision history
hm	18. oct. 2008	rev 1.0
	original version


*)

          
END_FUNCTION

FUNCTION BIT_LOAD_W : WORD
  VAR_INPUT
    IN : WORD;
    VAL : BOOL;
    POS : INT;
  END_VAR
  VAR CONSTANT
    dat : WORD := 1;
  END_VAR

            IF val THEN
	BIT_LOAD_W := in OR SHL(dat,pos);
ELSE
	BIT_LOAD_W := in AND (NOT SHL(dat,pos));
END_IF;


(* revision history
hm	29. feb 2008	rev 1.0
	original version

hm	16. mar 2008	rev 1.1
	change input bit to val for compatibility reasons
*)

          
END_FUNCTION

FUNCTION BIT_LOAD_W2 : WORD
  VAR_INPUT
    I : WORD;
    D : BOOL;
    P : INT;
    N : INT;
  END_VAR

            IF D THEN
	BIT_LOAD_W2 := ROL(SHR(WORD#65535, 16 - N) OR ROR(i, P), P);
ELSE
	BIT_LOAD_W2 := ROL(SHL(WORD#65535, N) AND ROR(I, P), P);
END_IF;



(* revision history
hm	18. oct. 2008	rev 1.0
	original version


*)

          
END_FUNCTION

FUNCTION BIT_OF_DWORD : BOOL
  VAR_INPUT
    in : DWORD;
    N : INT;
  END_VAR

            BIT_OF_DWORD := (SHR(in,N) AND 16#00000001) > 0;


(* old code used before rev 1.1
temp := SHR(in,n);
Bit_of_Dword := temp.0;
*)


(* revision history
hm	4. aug. 2006	rev 1.0
	original version

hm	29. feb 2008	rev 1.1
	improved performance

hm	6. jun. 2008	rev 1.2
	changes type of input N from byte to int
*)

          
END_FUNCTION

FUNCTION BIT_TOGGLE_B : BYTE
  VAR_INPUT
    IN : BYTE;
    POS : INT;
  END_VAR

            BIT_TOGGLE_B := SHL(BYTE#1, POS) XOR IN;




(* revision history
hm	18. oct. 2008	rev 1.0
	original version


*)

          
END_FUNCTION

FUNCTION BIT_TOGGLE_DW : DWORD
  VAR_INPUT
    IN : DWORD;
    POS : INT;
  END_VAR

            BIT_TOGGLE_DW := SHL(DWORD#1, POS) XOR IN;



(* revision history
hm	18. oct. 2008	rev 1.0
	original version


*)

          
END_FUNCTION

FUNCTION BIT_TOGGLE_W : WORD
  VAR_INPUT
    IN : WORD;
    POS : INT;
  END_VAR

            BIT_TOGGLE_W := SHL(WORD#1, POS) XOR IN;



(* revision history
hm	18. oct. 2008	rev 1.0
	original version


*)

          
END_FUNCTION

FUNCTION BYTE_OF_BIT : BYTE
  VAR_INPUT
    B0 : BOOL;
    B1 : BOOL;
    B2 : BOOL;
    B3 : BOOL;
    B4 : BOOL;
    B5 : BOOL;
    B6 : BOOL;
    B7 : BOOL;
  END_VAR

            Byte_of_bit := SHL(SHL(SHL(SHL(SHL(SHL(SHL(BOOL_TO_BYTE(B7),1) OR BOOL_TO_BYTE(B6),1) OR BOOL_TO_BYTE(B5),1) OR BOOL_TO_BYTE(B4),1)
	OR BOOL_TO_BYTE(B3),1) OR BOOL_TO_BYTE(B2),1) OR BOOL_TO_BYTE(B1),1) OR BOOL_TO_BYTE(B0);


(* revision history

hm	4. aug 2006		rev 1.0
	original version

hm	18. feb. 2008	rev 1.1
	improved performance

*)
          
END_FUNCTION

FUNCTION BYTE_OF_DWORD : BYTE
  VAR_INPUT
    in : DWORD;
    N : BYTE;
  END_VAR

            BYTE_OF_DWORD := DWORD_TO_BYTE(SHR(in,SHL(n,3)));

(* revision history
hm	17. jan 2007	rev 1.0
	original version

hm	2. jan 2008		rev 1.1
	improved performance

hm	30. oct. 2008	rev 1.2
	improved performance
*)


          
END_FUNCTION

FUNCTION_BLOCK BYTE_TO_BITS
  VAR_INPUT
    IN : BYTE;
  END_VAR
  VAR_OUTPUT
    B0 : BOOL;
    B1 : BOOL;
    B2 : BOOL;
    B3 : BOOL;
    B4 : BOOL;
    B5 : BOOL;
    B6 : BOOL;
    B7 : BOOL;
  END_VAR

            B0 := IN.0;
B1 := IN.1;
B2 := IN.2;
B3 := IN.3;
B4 := IN.4;
B5 := IN.5;
B6 := IN.6;
B7 := IN.7;

(* revision history
hm		4. aug 2006	rev 1.0
	original version

hm		16. mar 2008	rev 1.1
	renamed from byte_to_bit to byte_to_bits for compatibility reasons

*)
          
END_FUNCTION_BLOCK

FUNCTION BYTE_TO_GRAY : BYTE
  VAR_INPUT
    IN : BYTE;
  END_VAR

            BYTE_TO_GRAY := IN XOR SHR(IN,1);

(* revision history
hm	9. nov. 2009	rev 1.0
	original version

*)
          
END_FUNCTION

FUNCTION CHECK_PARITY : BOOL
  VAR_INPUT
    in : DWORD;
    p : BOOL;
  END_VAR

            CHECK_PARITY := NOT p;
WHILE in > 0 DO
	CHECK_PARITY := CHECK_PARITY XOR in.0 XOR in.1 XOR in.2 XOR in.3;
	in := SHR(in,4);
END_WHILE;

(* code before rev 1.2
WHILE in > 0 DO
	IF in.0 THEN cnt := cnt + 1; END_IF;
	in := SHR(in,1);
END_WHILE;
check_parity := even(cnt) XOR P;
*)


(* revision history

rev 1.0 HM  1.oct.2006

rev 1.1 hm	10.sep.2007
	changed algorithm to improove performance

rev 1.2	hm	8 dec 2007
	changed algorithm to improove performance

rev 1.3 hm	18. feb 2008
	changed algorithm to improove performance
*)
          
END_FUNCTION

FUNCTION CHK_REAL : BYTE
  VAR_INPUT
    X : REAL;
  END_VAR
  VAR
    pt : POINTER TO DWORD;
    tmp : DWORD;
  END_VAR

            pt := ADR(X);				(* move real to dword, real_to_dword does not work becasze it treats dword as a number on many systems *)
tmp := ROL(pt^,1);			(* rotate left foir easy checking, sign will be at lease significant digit *)
IF tmp < 16#FF000000 THEN
	CHK_REAL := 16#00;		(* normalized and denormalized numbers *)
ELSIF tmp = 16#FF000000 THEN
	CHK_REAL := 16#20;		(* X is +infinity see IEEE754 *)
ELSIF tmp = 16#FF000001 THEN
	CHK_REAL := 16#40;		(* X is -infinity see IEEE754 *)
ELSE
	CHK_REAL := 16#80;		(* X is NAN see IEEE754 *)
END_IF;


(* revision history
hm	 20. jan. 2011	rev 1.0
	original version

*)
          
END_FUNCTION

FUNCTION_BLOCK DEC_2
  VAR_INPUT
    D : BOOL;
    A : BOOL;
  END_VAR
  VAR_OUTPUT
    Q0 : BOOL;
    Q1 : BOOL;
  END_VAR

            Q0 := D AND NOT A;
Q1 := D AND A;

(* revision history
hm 3.3.2007	rev 1.1
	rewritten in ST for better compatibility

*)
          
END_FUNCTION_BLOCK

FUNCTION_BLOCK DEC_4
  VAR_INPUT
    D : BOOL;
    A0 : BOOL;
    A1 : BOOL;
  END_VAR
  VAR_OUTPUT
    Q0 : BOOL;
    Q1 : BOOL;
    Q2 : BOOL;
    Q3 : BOOL;
  END_VAR

            Q0 := D AND NOT A0 AND NOT A1;
Q1 := D AND A0 AND NOT A1;
Q2 := D AND NOT A0 AND A1;
Q3 := D AND A0 AND A1;

(* revision history
hm 3.3.2007	rev 1.1
	rewritten in ST for better compatibility

*)
          
END_FUNCTION_BLOCK

FUNCTION_BLOCK DEC_8
  VAR_INPUT
    D : BOOL;
    A0 : BOOL;
    A1 : BOOL;
    A2 : BOOL;
  END_VAR
  VAR_OUTPUT
    Q0 : BOOL;
    Q1 : BOOL;
    Q2 : BOOL;
    Q3 : BOOL;
    Q4 : BOOL;
    Q5 : BOOL;
    Q6 : BOOL;
    Q7 : BOOL;
  END_VAR
  VAR
    X : INT;
  END_VAR

            X.0 := A0; X.1 := A1; X.2 := A2;

Q0 := FALSE;
Q1 := FALSE;
Q2 := FALSE;
Q3 := FALSE;
Q4 := FALSE;
Q5 := FALSE;
Q6 := FALSE;
Q7 := FALSE;

CASE X OF
	0 : Q0 := D;
	1 : Q1 := D;
	2 : Q2 := D;
	3 : Q3 := D;
	4 : Q4 := D;
	5 : Q5 := D;
	6 : Q6 := D;
	7 : Q7 := D;
END_CASE;



(* revision history
hm 3. mar. 2007	rev 1.1
	rewritten in ST for better compatibility

hm	26. oct. 2008	rev 1.2
	code optimized

hm	28. mar. 2009	rev 1.3
	replaced multiple assignments
*)
          
END_FUNCTION_BLOCK

FUNCTION DW_TO_REAL : REAL
  VAR_INPUT
    X : DWORD;
  END_VAR
  VAR
    pt : POINTER TO REAL;
  END_VAR

            pt := ADR(X);
DW_TO_REAL := pt^;

(* revision history
hm	18. apr. 2008
	original version

*)
          
END_FUNCTION

FUNCTION DWORD_OF_BYTE : DWORD
  VAR_INPUT
    B3 : BYTE;
    B2 : BYTE;
    B1 : BYTE;
    B0 : BYTE;
  END_VAR

            DWORD_OF_BYTE := SHL(SHL(SHL(BYTE_TO_DWORD(B3),8) OR BYTE_TO_DWORD(B2),8) OR BYTE_TO_DWORD(B1),8) OR BYTE_TO_DWORD(B0);


(* revision history
hm	24. jan 2007	rev 1.0
	original version

hm 2. jan 2008	rev 1.1
	inproved performance

hm	23. apr. 2008	rev 1.2
	reverse order of inputs to be more logical

hm	18. jul. 2009	rev 1.3
	added type conversions for compatibility reasons
*)
          
END_FUNCTION

FUNCTION DWORD_OF_WORD : DWORD
  VAR_INPUT
    W1 : WORD;
    W0 : WORD;
  END_VAR

            DWORD_OF_WORD := SHL(WORD_TO_DWORD(W1),16) OR WORD_TO_DWORD(W0);


(* revision history

hm	18. jul. 2009	rev 1.0
	original version

*)
          
END_FUNCTION

FUNCTION GRAY_TO_BYTE : BYTE
  VAR_INPUT
    IN : BYTE;
  END_VAR

            GRAY_TO_BYTE := SHR(IN,4) XOR IN;
GRAY_TO_BYTE := SHR(GRAY_TO_BYTE,2) XOR GRAY_TO_BYTE;
GRAY_TO_BYTE := SHR(GRAY_TO_BYTE,1) XOR GRAY_TO_BYTE;

(* revision history
hm	9. nov. 2009	rev 1.0
	original version

*)
          
END_FUNCTION

FUNCTION INT_TO_BCDC : BYTE
  VAR_INPUT
    IN : INT;
  END_VAR

            INT_TO_BCDC := SHL(INT_TO_BYTE(IN / INT#10),4) OR INT_TO_BYTE(in MOD INT#10);

(* revision history
hm	13.12.2007
	original version

hm	30.6.2008	rev 1.1
	changed name INT_TO_BCD to INT_TO_BCDC to avoid collision with util.lib
	corrected error in code

*)
          
END_FUNCTION

FUNCTION MUX_2 : BOOL
  VAR_INPUT
    D0 : BOOL;
    D1 : BOOL;
    A0 : BOOL;
  END_VAR

            MUX_2 := SEL(A0, D0, D1);


(*
revision history:
hm	5.10.2006		rev 1.1
	changed to ST Langage for better portability.

hm	16. oct. 2008	rev 1.2
	improved performance

*)
          
END_FUNCTION

FUNCTION MUX_4 : BOOL
  VAR_INPUT
    D0 : BOOL;
    D1 : BOOL;
    D2 : BOOL;
    D3 : BOOL;
    A0 : BOOL;
    A1 : BOOL;
  END_VAR

            IF A1 THEN
	MUX_4 := SEL(A0, D2, D3);
ELSE
	MUX_4 := SEL(A0, D0, D1);
END_IF;


(*
revision history:
hm 	5.10.2006		rev 1.1
	rewritten to ST for better portability

hm	16. oct. 2008	rev 1.2
	improved performance

*)
          
END_FUNCTION

FUNCTION PARITY : BOOL
  VAR_INPUT
    in : DWORD;
  END_VAR

            WHILE in > 0 DO
	PARITY := PARITY XOR in.0 XOR in.1 XOR in.2 XOR in.3;
	in := SHR(in,4);
END_WHILE;

(* code before rev 1.2
WHILE in > 0 DO
	IF in.0 THEN cnt := cnt +1; END_IF;
	in := SHR(in,1);
END_WHILE;
IF (cnt MOD 2) = 1 THEN parity := TRUE; ELSE parity := FALSE; END_IF;
*)

(* revision history

rev 1.0 hm 1 sep 2006
	original version

rev 1.1 hm 10.9.2007
	changed algorithm to improve performance

rev 1.2	hm	8 dec 2007
	changed algorithm to improve performance

rev 1.3	hm	18 feb 2008
	changed algorithm to improve performance
*)
          
END_FUNCTION

FUNCTION REAL_TO_DW : DWORD
  VAR_INPUT
    X : REAL;
  END_VAR
  VAR
    pt : POINTER TO DWORD;
  END_VAR

            pt := ADR(X);
REAL_TO_DW := pt^;

(* revision history
hm	18. apr. 2008
	original version

*)
          
END_FUNCTION

FUNCTION REFLECT : DWORD
  VAR_INPUT
    D : DWORD;
    L : INT;
  END_VAR
  VAR
    i : INT;
  END_VAR

            REFLECT := 0;
FOR i := 1 TO L DO
	REFLECT := SHL(REFLECT, 1) OR BOOL_TO_DWORD(D.0);
	D := SHR(D, 1);
END_FOR;
REFLECT := REFLECT OR SHL(D, L);

(* revision history
hm	 16. jan 2011
	new module

*)
          
END_FUNCTION

FUNCTION REVERSE : BYTE
  VAR_INPUT
    IN : BYTE;
  END_VAR

            REVERSE := SHL(in,7) OR SHR(in,7) OR (ROR(in,3) AND 2#01000100) OR (ROL(in,3) AND 2#00100010)
	OR (SHL(in,1) AND 2#00010000) OR (SHR(in,1) AND 2#00001000);


(* revision history
hm		9.oct 2007		rev 1.0
	original version

hm		18. feb 2008	rev 1.1
	improved performance
*)
          
END_FUNCTION

FUNCTION SHL1 : DWORD
  VAR_INPUT
    IN : DWORD;
    N : INT;
  END_VAR
  VAR CONSTANT
    temp : DWORD := 16#FFFFFFFF;
  END_VAR

            SHL1 := SHR(temp,32-N) OR SHL(IN,N);


(* revision history
hm	14.9.2007		rev 1.0
	original version

hm	27. dec 2007	rev 1.1
	changed code for better performance

*)
          
END_FUNCTION

FUNCTION SHR1 : DWORD
  VAR_INPUT
    IN : DWORD;
    N : INT;
  END_VAR
  VAR CONSTANT
    temp : DWORD := 16#FFFFFFFF;
  END_VAR

            SHR1 := SHL(temp,32-N) OR SHR(IN,N);

(* revision history
hm	14.9.2007		rev 1.0
	original version

hm	27. dec 2007	rev 1.1
	changed code for better performance

*)
          
END_FUNCTION

FUNCTION SWAP_BYTE : WORD
  VAR_INPUT
    IN : WORD;
  END_VAR

            SWAP_BYTE := ROL(in,8);


(* revision history
hm		4. feb 2008	rev 1.0
	original version

*)
          
END_FUNCTION

FUNCTION SWAP_BYTE2 : DWORD
  VAR_INPUT
    IN : DWORD;
  END_VAR

            Swap_Byte2 := (ROR(in,8) AND 16#FF00FF00) OR (ROL(in,8) AND 16#00FF00FF);

(* revision history
hm		4. feb 2008	rev 1.0
	original version

*)

          
END_FUNCTION

FUNCTION WORD_OF_BYTE : WORD
  VAR_INPUT
    B1 : BYTE;
    B0 : BYTE;
  END_VAR

            WORD_OF_BYTE := SHL(BYTE_TO_WORD(B1),8) OR BYTE_TO_WORD(B0);

(* revision history
hm	24. jan 2007	rev 1.0
	original version

hm	2. jan 2008	rev 1.1
	improved performance

hm	19. feb 2008	rev 1.2
	replaced and with or for better compatibility

hm	23. apr. 2008	rev 1.3
	reverse order of inputs to be more logical

hm	18. jul. 2009	rev 1.4
	added type conversions for compatibility reasons

*)
          
END_FUNCTION

FUNCTION WORD_OF_DWORD : WORD
  VAR_INPUT
    in : DWORD;
    N : BYTE;
  END_VAR

            WORD_OF_DWORD := DWORD_TO_WORD(SHR(in,SHL(n,4)));

(* revision history
hm	17. jan 2007	rev 1.0
	original version

hm	2. jan 2008		rev 1.1
	improved performance

hm	30. oct. 2008	rev 1.2
	improved performance
*)

          
END_FUNCTION

FUNCTION_BLOCK A_TRIG
  VAR_INPUT
    IN : REAL;
    RES : REAL;
  END_VAR
  VAR_OUTPUT
    Q : BOOL;
    D : REAL;
  END_VAR
  VAR
    last_in : REAL;
  END_VAR

            D := IN - LAST_IN;
Q := ABS(D) > res;
IF Q THEN last_in := IN; END_IF;
D := IN - LAST_IN;


(* revision history

hm 	16. jul. 2008	rev 1.0
	original version released

hm	25. oct. 2008	rev 1.1
	code optimization
	a_trig now also works for res = 0

*)
          
END_FUNCTION_BLOCK

FUNCTION_BLOCK B_TRIG
  VAR_INPUT
    CLK : BOOL;
  END_VAR
  VAR_OUTPUT
    Q : BOOL;
  END_VAR
  VAR
    edge : BOOL;
  END_VAR

            Q := clk XOR edge;
edge := CLK;


(* revision history
hm		4. aug. 2006	rev 1.0
	original version

*)
          
END_FUNCTION_BLOCK

FUNCTION_BLOCK CLICK_CNT
  VAR_INPUT
    IN : BOOL;
    N : INT;
    TC : TIME;
  END_VAR
  VAR_OUTPUT
    Q : BOOL;
  END_VAR
  VAR
    tx : TP;
    edge : BOOL;
    cnt : INT := -1;
  END_VAR

            (* Q shall only be active for one cycle only *)
Q := FALSE;

IF in AND NOT edge AND NOT tx.q THEN
	(* a rising edge on in sets the counter to 0 *)
	cnt := 0;
ELSIF tx.Q AND NOT IN AND edge THEN
	(* count falling edges when tp.q is true *)
	cnt := cnt + 1;
ELSIF NOT tx.Q THEN
	Q := cnt = N;
	cnt := -1;
END_IF;

(* remember the status of IN *)
edge := IN;
tx(in := IN, pt := TC);


(* revision history

hm 	16. jul. 2008	rev 1.0
	original version released


*)
          
END_FUNCTION_BLOCK

FUNCTION_BLOCK CLICK_DEC
  VAR_INPUT
    IN : BOOL;
    TC : TIME;
  END_VAR
  VAR_OUTPUT
    Q0 : BOOL;
    Q1 : BOOL;
    Q2 : BOOL;
    Q3 : BOOL;
  END_VAR
  VAR
    tx : TP;
    edge : BOOL;
    cnt : INT := -1;
  END_VAR

            (* Q shall only be active for one cycle only *)
IF in = FALSE THEN
	Q0 := FALSE;
	Q1 := FALSE;
	Q2:= FALSE;
	Q3 := FALSE;
END_IF;

IF in AND NOT edge AND NOT tx.q THEN
	(* a rising edge on in sets the counter to 0 *)
	cnt := 0;
ELSIF tx.Q AND NOT IN AND edge THEN
	(* count falling edges when tp.q is true *)
	cnt := cnt + 1;
ELSIF NOT tx.Q THEN
	CASE cnt OF
		0 : Q0 := TRUE;
		1 : Q1 := TRUE;
		2 : Q2 := TRUE;
		3 : Q3 := TRUE;
	END_CASE;
	cnt := -1;
END_IF;

(* remember the status of IN *)
edge := IN;
tx(in := IN, pt := TC);



(* revision history

hm 17. jul. 2008	rev 1.0
	original version released

hm	14. mar. 2009	rev 1.1
	removed double assignments

*)
          
END_FUNCTION_BLOCK

FUNCTION_BLOCK CLK_DIV
  VAR_INPUT
    clk : BOOL;
    rst : BOOL;
  END_VAR
  VAR_OUTPUT
    Q0 : BOOL;
    Q1 : BOOL;
    Q2 : BOOL;
    Q3 : BOOL;
    Q4 : BOOL;
    Q5 : BOOL;
    Q6 : BOOL;
    Q7 : BOOL;
  END_VAR
  VAR
    cnt : BYTE;
  END_VAR

            IF rst THEN
	cnt:= 0;
	Q0 := 0;
	Q1 := 0;
	Q2 := 0;
	Q3 := 0;
	Q4 := 0;
	Q5 := 0;
	Q6 := 0;
	Q7 := 0;
ELSIF clk THEN
	cnt:= cnt +1;
	Q0 := cnt.0;
	Q1 := cnt.1;
	Q2 := cnt.2;
	Q3 := cnt.3;
	Q4 := cnt.4;
	Q5 := cnt.5;
	Q6 := cnt.6;
	Q7 := cnt.7;
END_IF;

(* revision history
hm	4. aug. 2006	rev 1.0
	original version

hm	2. jan 2008		rev 1.1
	improved performance

*)
          
END_FUNCTION_BLOCK

FUNCTION_BLOCK CLK_N
  VAR_INPUT
    N : INT;
  END_VAR
  VAR_OUTPUT
    Q : BOOL;
  END_VAR
  VAR
    edge : BOOL;
    stime : DWORD;
    clk : BOOL;
  END_VAR

            stime := SHR(T_PLC_MS(),N);
clk := stime.0;
Q := clk XOR edge;
edge := CLK;

(* revision history
hm	16. dec 2007		rev 1.0
	original version

*)
          
END_FUNCTION_BLOCK

FUNCTION_BLOCK CLK_PRG
  VAR_INPUT
    PT : TIME := TIME#10ms;
  END_VAR
  VAR_OUTPUT
    Q : BOOL;
  END_VAR
  VAR
    init : BOOL;
    last : TIME;
    tx : TIME;
  END_VAR

            (* read system time *)
tx := DWORD_TO_TIME(T_PLC_MS());

(* initialize on startup *)
IF NOT init THEN
	init := TRUE;
	last := tx - pt;
END_IF;

(* generate output pulse when next_pulse is reached *)
Q := tx - last >= pt;
IF Q THEN last := tx; END_IF;


(* revision hiostory

hm 25 feb 2007	rev 1.1
	rewritten code for higher performance
	pt can now be changed during runtime

hm	17. sep 2007	rev 1.2
	replaced time() with t_plc_ms() for compatibility reasons

hm	25. oct. 2008	rev 1.3
	optimized code

*)
          
END_FUNCTION_BLOCK

FUNCTION_BLOCK CLK_PULSE
  VAR_INPUT
    PT : TIME;
    N : INT;
    RST : BOOL;
  END_VAR
  VAR_OUTPUT
    Q : BOOL;
    CNT : INT;
    RUN : BOOL;
  END_VAR
  VAR
    tx : DWORD;
    tn : DWORD;
    init : BOOL;
  END_VAR

            tx := T_PLC_MS();		(* read system *)
Q := FALSE;				(* reset Q we generate pulses only for one cycle *)
RUN := CNT < N;

IF NOT init OR RST THEN
	init := TRUE;
	CNT := 0;
	tn := tx - TIME_TO_DWORD(PT);
	RUN := FALSE;
ELSIF (cnt < N OR N = 0) AND tx - tn >= TIME_TO_DWORD(PT) THEN		(* generate a pulse *)
	CNT := CNT + 1;
	Q := TRUE;
	tn := tn + TIME_TO_DWORD(PT);
END_IF;



(* revision history
hm		4. aug 2006		rev 1.0
	original version

hm		17. sep 2007	rev 1.1
	replaced time() with T_PLC_S() for compatblity reasons

hm		16. feb. 2011	rev 1.2
	fixed an error when timer overflows 
*)
          
END_FUNCTION_BLOCK

FUNCTION_BLOCK CYCLE_4
  VAR_INPUT
    E : BOOL := TRUE;
    T0 : TIME;
    T1 : TIME;
    T2 : TIME;
    T3 : TIME;
    S0 : BOOL;
    SX : INT;
    SL : BOOL;
  END_VAR
  VAR_OUTPUT
    STATE : INT;
  END_VAR
  VAR
    tx : TIME;
    last : TIME;
    init : BOOL;
  END_VAR

            (* read system timer *)
tx := DWORD_TO_TIME(T_PLC_MS());
(* init on first cycle *)
IF NOT init THEN
	init := TRUE;
	last := tx;
END_IF;

IF E THEN
	IF SL THEN
		(* when sx > 0 then the state sx is forced to start *)
		state:= LIMIT(0,SX,3);
		last := tx;
		(* this is to avoid to reset sx from the calling programm it does work fine on codesys but i am not sure about other systems, because we are writing to an input *)
		SL := FALSE;
	ELSE
		CASE state OF
			0 :	(* wait for T0 and switch to next cycle *)
				IF tx - last >= T0 THEN
					state := 1;
					last := tx;
				END_IF;
			1 : (* wait for T1 over 1st cycle *)
				IF tx - last >= T1 THEN
					state := 2;
					last := tx;
				END_IF;
			2 : (* wait for T1 over 1st cycle *)
				IF tx - last >= T2 THEN
					state := 3;
					last := tx;
				END_IF;
			3 : (* wait for T2 over 2nd cycle *)
				IF tx - last >= T3 THEN
					IF S0 THEN State := 0; END_IF; (* if S0 is false, the sequence stops at state 3 *)
					last := tx;
				END_IF;
		END_CASE;
	END_IF;
ELSE
	state := 0;
	last := tx;
END_IF;



(*
hm	3. nov. 2008	rev 1.0
	original version

*)
          
END_FUNCTION_BLOCK

FUNCTION_BLOCK D_TRIG
  VAR_INPUT
    in : DWORD;
  END_VAR
  VAR_OUTPUT
    Q : BOOL;
    X : DWORD;
  END_VAR
  VAR
    last_in : DWORD;
  END_VAR

            Q := in <> last_in;
X := in - last_in;
last_in := in;


(* revision history

hm 	4.09.2007		rev 1.0
	original version released

hm	19. feb. 2008	rev 1.1
	performance improvement
*)
          
END_FUNCTION_BLOCK

FUNCTION_BLOCK GEN_BIT
  VAR_INPUT
    in0 : DWORD;
    in1 : DWORD;
    in2 : DWORD;
    in3 : DWORD;
    clk : BOOL;
    steps : INT;
    rep : INT;
    rst : BOOL;
  END_VAR
  VAR_OUTPUT
    Q0 : BOOL;
    Q1 : BOOL;
    Q2 : BOOL;
    Q3 : BOOL;
    cnt : INT;
    run : BOOL;
  END_VAR
  VAR
    r0 : DWORD;
    r1 : DWORD;
    r2 : DWORD;
    r3 : DWORD;
    rx : INT := 1;
  END_VAR

            (* check if number of runs is finished or rep = 0 which means continuous *)

IF clk AND NOT rst THEN
	run := (rep = 0) OR (rx <= rep);
	IF run THEN
		(* check for step counter reached and reset to 0 if cnt = steps *)
		IF cnt = steps THEN
			cnt := 0;
		END_IF;

		(* when cnt = 0 then reload the inputs into the registers *)
		IF cnt = 0 THEN
			r0 := in0;
			r1 := in1;
			r2 := in2;
			r3 := in3;
		END_IF;

		(* when cnt < steps, shift the lowest bits to the outputs *)
		IF (cnt < steps) THEN
			Q0 := r0.0;
			Q1 := r1.0;
			Q2 := r2.0;
			Q3 := r3.0;
			r0 := SHR(r0,1);
			r1 := SHR(r1,1);
			r2 := SHR(r2,1);
			r3 := SHR(r3,1);
		END_IF;

		(* increment the step counter *)
		cnt := cnt +1;
		IF (cnt = steps) AND (rep <> 0) THEN rx := rx +1; END_IF;
		IF (rx > rep) AND (rep <> 0) THEN run := FALSE; END_IF;
	END_IF;
ELSE
	IF rst THEN
		run := FALSE;
		Q0 := FALSE;
		Q1 := FALSE;
		Q2 := FALSE;
		Q3 := FALSE;
		r0 := 0;
		r1 := 0;
		r2 := 0;
		r3 := 0;
		cnt := 0;
		rx := 1;
	END_IF;
END_IF;



(* revision histroy
hm	4 aug 2006	rev 1.0
	original version

hm 15. oct. 2008	rev 1.1
	improved performance

hm	14. mar. 2009	rev 1.2
	removed double assignments

*)
          
END_FUNCTION_BLOCK

FUNCTION_BLOCK GEN_SQ
  VAR_INPUT
    PT : TIME;
  END_VAR
  VAR_OUTPUT
    Q : BOOL;
  END_VAR
  VAR
    tn : DWORD;
    tx : DWORD;
    init : BOOL;
  END_VAR

            (* read system time *)
tx := T_PLC_MS();

IF NOT init THEN
	init := TRUE;
	tn := tx;
	Q := TRUE;
ELSIF tx - tn >= SHR(TIME_TO_DWORD(PT),1) THEN
	Q := NOT Q;
	tn := tn + SHR(TIME_TO_DWORD(pt),1);
END_IF;


(* revision history
hm	4. aug 2006	rev 1.0
	original version

hm	17. sep 2007	rev 1.1
	replaced time() with T_PLC_MS() for compatibility reasons

hm	18. jul. 2009	rev 1.2
	improved accuracy

hm	16. feb 2011	rev 1.3
	corrected an error with timer overflow 
*)




          
END_FUNCTION_BLOCK

FUNCTION_BLOCK SCHEDULER
  VAR_INPUT
    E0 : BOOL;
    E1 : BOOL;
    E2 : BOOL;
    E3 : BOOL;
    {attribute 'input_constant'}
    T0 : TIME;
    {attribute 'input_constant'}
    T1 : TIME;
    {attribute 'input_constant'}
    T2 : TIME;
    {attribute 'input_constant'}
    T3 : TIME;
  END_VAR
  VAR_OUTPUT
    Q0 : BOOL;
    Q1 : BOOL;
    Q2 : BOOL;
    Q3 : BOOL;
  END_VAR
  VAR
    init : BOOL;
    s0 : TIME;
    s1 : TIME;
    s2 : TIME;
    s3 : TIME;
    tx : TIME;
    c : INT;
  END_VAR

            (* read system_time *)
tx := DWORD_TO_TIME(T_PLC_MS());

IF NOT init THEN
	init := TRUE;
	s0 := tx - T0;
	s1 := tx - T1;
	s2 := tx - T2;
	s3 := tx - T3;
END_IF;

Q0 := FALSE;
Q1 := FALSE;
Q2 := FALSE;
Q3 :=FALSE;

CASE c OF
	0: 	IF tx - s0 >= T0 THEN
			Q0 := E0;
			s0 := tx;
		END_IF;
		c := 1;
	1: 	IF tx - s1 >= T1 THEN
			Q1 := E1;
			s1 := tx;
		END_IF;
		c := 2;
	2: 	IF tx - s2 >= T2 THEN
			Q2 := E2;
			s2 := tx;
		END_IF;
		c := 3;
	3: 	IF tx - s3 >= T3 THEN
			Q3 := E3;
			s3 := tx;
		END_IF;
		c := 0;
END_CASE;


(* revision history

hm 28. sep. 2008	rev 1.0
	original version

hm	14. mar. 2009	rev 1.1
	removed double assignments

*)
          
END_FUNCTION_BLOCK

FUNCTION_BLOCK SCHEDULER_2
  VAR_INPUT
    E0 : BOOL;
    E1 : BOOL;
    E2 : BOOL;
    E3 : BOOL;
    {attribute 'input_constant'}
    C0 : UINT;
    {attribute 'input_constant'}
    C1 : UINT;
    {attribute 'input_constant'}
    C2 : UINT;
    {attribute 'input_constant'}
    C3 : UINT;
    {attribute 'input_constant'}
    O0 : UINT;
    {attribute 'input_constant'}
    O1 : UINT;
    {attribute 'input_constant'}
    O2 : UINT;
    {attribute 'input_constant'}
    O3 : UINT;
  END_VAR
  VAR_OUTPUT
    Q0 : BOOL;
    Q1 : BOOL;
    Q2 : BOOL;
    Q3 : BOOL;
  END_VAR
  VAR
    sx : UINT;
  END_VAR

            Q0 := E0 AND (sx MOD C0 - O0 = 0);
Q1 := E1 AND (sx MOD C1 - O1 = 0);
Q2 := E2 AND (sx MOD C2 - O2 = 0);
Q3 := E3 AND (sx MOD C3 - O3 = 0);

(* increment cycle counter every cycle *)
sx := sx + 1;


(* revision history
hm 29. sep. 2008		rev 1.0
	original version


*)
          
END_FUNCTION_BLOCK

FUNCTION_BLOCK SEQUENCE_4
  VAR_INPUT
    in0 : BOOL := TRUE;
    in1 : BOOL := TRUE;
    in2 : BOOL := TRUE;
    in3 : BOOL := TRUE;
    start : BOOL;
    rst : BOOL;
    wait0 : TIME;
    delay0 : TIME;
    wait1 : TIME;
    delay1 : TIME;
    wait2 : TIME;
    delay2 : TIME;
    wait3 : TIME;
    delay3 : TIME;
    {attribute 'input_constant'}
    stop_on_error : BOOL;
  END_VAR
  VAR_OUTPUT
    Q0 : BOOL;
    Q1 : BOOL;
    Q2 : BOOL;
    Q3 : BOOL;
    QX : BOOL;
    run : BOOL;
    step : INT := -1;
    status : BYTE;
  END_VAR
  VAR
    last : TIME;
    edge : BOOL;
    tx : TIME;
    init : BOOL;
  END_VAR

            (* read sps timer *)
tx := DWORD_TO_TIME(T_PLC_MS());

(* initialize on startup *)
IF NOT init THEN
	last := tx;
	init := TRUE;
	status := 110;
END_IF;

(* asynchronous reset *)
IF rst THEN
	step := -1;
	Q0 := 0;
	Q1 := 0;
	Q2 := 0;
	Q3 := 0;
	status := 110;
	run := 0;

(* edge on start input restarts the sequencer *)
ELSIF start AND NOT edge THEN
	step := 0;
	last := tx;
	status := 111;
	Q0 := 0;
	Q1 := 0;
	Q2 := 0;
	Q3 := 0;
	run := 1;
END_IF;
edge := start;

(* check if stop on status is necessary *)
IF status > 0 AND status < 100 AND stop_on_error THEN RETURN; END_IF;

(* sequence is running *)
IF run AND step = 0 THEN
	IF NOT q0 AND in0 AND tx - last <= wait0 THEN
		Q0 := TRUE;
		last := tx;
	ELSIF NOT q0 AND tx - last > wait0 THEN
		status := 1;
		run := FALSE;
	ELSIF q0 AND tx - last >= delay0 THEN
		step := 1;
		last := tx;
	END_IF;
END_IF;
IF run AND step = 1 THEN
	IF NOT q1 AND in1 AND tx - last <= wait1 THEN
		Q0 := FALSE;
		Q1 := TRUE;
		last := tx;
	ELSIF NOT q1 AND Tx - last > wait1 THEN
		status := 2;
		q0 := FALSE;
		run := FALSE;
	ELSIF q1 AND tx - last >= delay1 THEN
		step := 2;
		last := tx;
	END_IF;
END_IF;
IF run AND step = 2 THEN
	IF NOT q2 AND in2 AND tx - last <= wait2 THEN
		Q1 := FALSE;
		Q2 := TRUE;
		last := tx;
	ELSIF NOT q2 AND Tx - last > wait2 THEN
		status := 3;
		q1 := FALSE;
		run := FALSE;
	ELSIF q2 AND tx - last >= delay2 THEN
		step := 3;
		last := tx;
	END_IF;
END_IF;
IF run AND step = 3 THEN
	IF NOT q3 AND in3 AND tx - last <= wait3 THEN
		Q2 := FALSE;
		Q3 := TRUE;
		last := tx;
	ELSIF NOT q3 AND Tx - last > wait3 THEN
		status := 4;
		q2 := FALSE;
		run := FALSE;
	ELSIF q3 AND tx - last >= delay3 THEN
		step := -1;
		q3 := FALSE;
		run := FALSE;
		status := 110;
	END_IF;
END_IF;
QX := q0 OR q1 OR q2 OR q3;

(*
hm 1.10.06		rev 1.1
	corrected delay logic to be after event and not before
	added any output

hm 1.12.06		rev 1.2
	corrected failure in sequence logic.
	added init at startup to prevent from initial error after start.

hm 17.1.2007		rev 1.3
	changed output fault to status for better compatibility with other modules (ESR).
	added stop on error functionality and setup variable
	default for inputs in0..3 is true.
	renamed variable state to step

hm	17.sep 2007	rev 1.4
	replaced time() with T_PLC_MS() for compatibility reasons

hm	13. mar. 2009	rev 1.5
	renamed output any to qx for compatibility resons

*)
          
END_FUNCTION_BLOCK

FUNCTION_BLOCK SEQUENCE_64
  VAR_INPUT
    START : BOOL;
    SMAX : INT;
    PROG : ARRAY[0..63] OF TIME;
    RST : BOOL;
  END_VAR
  VAR_OUTPUT
    STATE : INT := -1;
    TRIG : BOOL;
  END_VAR
  VAR
    tx : TIME;
    edge : BOOL;
    last : TIME;
  END_VAR

